KUKA KRL program: EPS_2_25252_SD6A_A_20250910061730.src

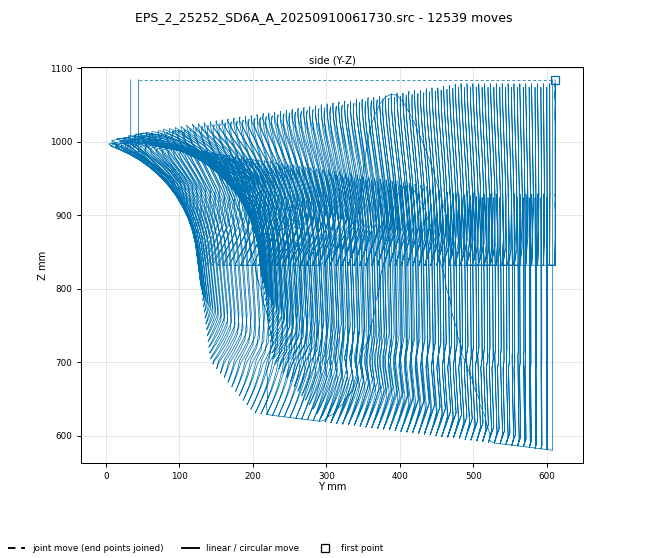
[picture p0: tool path of EPS_2_25252_SD6A_A_20250910061730.src, 12539 of 12541 moves have a stored position in this frame; points joined in program order, loops and branches not executed]
&ACCESS RVP
&REL 4
&COMMENT QRS 19112012
&PARAM EDITMASK = *
DEF PART()
EXT BAS (BAS_COMMAND :IN,REAL :IN )
INT I
BAS (#INITMOV,0 )

;KUKA QRS Post kuka4.cps  Date:22-06-2017 !

File_ID=2826

QRS_PRE_INIT()

;Init var - Until changes are made in qrs_pre_init
Outlet_Square_prg=0
Inlet_1_Square_prg=0
Inlet_2_Square_prg=0
Inlet_3_Square_prg=0
Inlet_4_Square_prg=0
Inlet_5_Square_prg=0

Outlet_1={X 0.000, Y 484.060, Z 891.000, B 0.000, E1 0.000 }
Inlet_1={X 0.000, Y 511.230, Z 798.500, B 0.000, E1 160.000 }
Outlet_1_type=366
Inlet_1_type=201
;QRS#1=Sidecore dimensions
;QRS#2=375-15" PVC SDR 35
;QRS#3=200-8" PVC SDR 35
;QRS#4=
;QRS#5=
;QRS#6=
;QRS#7=
;QRS#8=
;QRS#9=20Y PSX
;QRS#10=12-08 PSX
;QRS#11=
;QRS#12=
;QRS#13=
;QRS#14=
;QRS#15=
;QRS#16=1220x127x1372 4,5'
;QRS#17=EPS Height
;QRS#18=1074
;QRS#19=*
;QRS#20= UPDATED VERSION 22-06-2017
;QRS#21=*
Outlet_Square=0250
Inlet_1_Square=0100
Inlet_2_Square=0
Inlet_3_Square=0
Inlet_4_Square=0
Inlet_5_Square=0
Mill_Square=1
Outlet_Square_Prg=252
Inlet_1_Square_prg=204

QRS_INIT()

$ADVANCE=5

; T1
PTP {E1 177.357,E2 177.357}
PTP {X 0,Y 611.096,A -85,B 0,C 180,E1 177.357,E2 177.357,E3 0,E4 0,E5 0,E6 0}
QRS_SPEED_INIT()
LIN {X 0,Y 611.096,Z 1084,A -85,B 0,C 180,E1 177.357,E2 177.357,E3 0,E4 0,E5 0,E6 0} C_VEL
LIN {X 0,Y 611.096,Z 833.81,A -85,B 0,C 180,E1 177.357,E2 177.357} C_VEL
LIN {X 0,Y 611.169,Z 831.81,A -85,B 0,C 180,E1 177.544,E2 177.544} C_VEL
LIN {X 0,Y 611.846,Z 831.81,A -85,B 0,C 180,E1 178.833,E2 178.833} C_VEL
LIN {X 0,Y 611.842,Z 831.81,A -85,B 0,C 180,E1 185.845,E2 185.845} C_VEL
LIN {X 0,Y 611.87,Z 831.81,A -85,B 0,C 180,E1 192.946,E2 192.946} C_VEL
LIN {X 0,Y 611.805,Z 831.81,A -85,B 0,C 180,E1 200.259,E2 200.259} C_VEL
LIN {X 0,Y 611.785,Z 831.81,A -85,B 0,C 180,E1 207.936,E2 207.936} C_VEL
LIN {X 0,Y 610.448,Z 831.81,A -85,B 0,C 180,E1 210.686,E2 210.686} C_VEL
LIN {X 0,Y 611.751,Z 831.81,A -85,B 0,C 180,E1 216.209,E2 216.209} C_VEL
LIN {X 0,Y 611.181,Z 831.81,A -85,B 0,C 180,E1 217.329,E2 217.329} C_VEL
LIN {X 0,Y 610.711,Z 831.81,A -85,B 0,C 180,E1 222.327,E2 222.327} C_VEL
LIN {X 0,Y 611.733,Z 831.81,A -85,B 0,C 180,E1 224.523,E2 224.523} C_VEL
LIN {X 0,Y 611.705,Z 831.81,A -85,B 0,C 180,E1 232.607,E2 232.607} C_VEL
LIN {X 0,Y 611.184,Z 831.81,A -85,B 0,C 180,E1 233.752,E2 233.752} C_VEL
LIN {X 0,Y 611.693,Z 831.81,A -85,B 0,C 180,E1 241.163,E2 241.163} C_VEL
LIN {X 0,Y 611.503,Z 831.81,A -85,B 0,C 180,E1 242.05,E2 242.05} C_VEL
LIN {X 0,Y 611.8,Z 831.81,A -85,B 0,C 180,E1 248.625,E2 248.625} C_VEL
LIN {X 0,Y 610.992,Z 831.81,A -85,B 0,C 180,E1 248.983,E2 248.983} C_VEL
LIN {X 0,Y 610.765,Z 831.863,A -85,B 0,C 180,E1 249.009,E2 249.009} C_VEL
LIN {X 0,Y 611.59,Z 868.04,A -85,B 0,C 180,E1 249.483,E2 249.483} C_VEL
LIN {X 0,Y 611.819,Z 897.067,A -85,B 0,C 180,E1 249.858,E2 249.858} C_VEL
LIN {X 0,Y 611.837,Z 906.232,A -85,B 0,C 180,E1 250.014,E2 250.014} C_VEL
LIN {X 0,Y 611.813,Z 915.284,A -85,B 0,C 180,E1 250.207,E2 250.207} C_VEL
LIN {X 0,Y 611.665,Z 924.239,A -85,B 0,C 180,E1 250.435,E2 250.435} C_VEL
LIN {X 0,Y 611.793,Z 933.099,A -85,B 0,C 180,E1 250.71,E2 250.71} C_VEL
LIN {X 0,Y 611.793,Z 940.863,A -85,B 0,C 180,E1 250.98,E2 250.98} C_VEL
LIN {X 0,Y 611.788,Z 950.494,A -85,B 0,C 180,E1 251.365,E2 251.365} C_VEL
LIN {X 0,Y 611.804,Z 958.998,A -85,B 0,C 180,E1 251.75,E2 251.75} C_VEL
LIN {X 0,Y 611.728,Z 968.053,A -85,B 0,C 180,E1 252.208,E2 252.208} C_VEL
LIN {X 0,Y 611.708,Z 977.508,A -85,B 0,C 180,E1 252.747,E2 252.747} C_VEL
LIN {X 0,Y 611.545,Z 985.953,A -85,B 0,C 180,E1 253.278,E2 253.278} C_VEL
LIN {X 0,Y 611.448,Z 992.373,A -85,B 0,C 180,E1 253.719,E2 253.719} C_VEL
LIN {X 0,Y 611.514,Z 999.796,A -85,B 0,C 180,E1 254.279,E2 254.279} C_VEL
LIN {X 0,Y 611.73,Z 1007.694,A -85,B 0,C 180,E1 254.936,E2 254.936} C_VEL
LIN {X 0,Y 611.83,Z 1014.191,A -85,B 0,C 180,E1 255.523,E2 255.523} C_VEL
LIN {X 0,Y 611.643,Z 1021.1,A -85,B 0,C 180,E1 256.197,E2 256.197} C_VEL
LIN {X 0,Y 611.384,Z 1027.094,A -85,B 0,C 180,E1 256.831,E2 256.831} C_VEL
LIN {X 0,Y 611.257,Z 1032.807,A -85,B 0,C 180,E1 257.49,E2 257.49} C_VEL
LIN {X 0,Y 611.362,Z 1038.701,A -85,B 0,C 180,E1 258.239,E2 258.239} C_VEL
LIN {X 0,Y 611.558,Z 1043.069,A -85,B 0,C 180,E1 258.838,E2 258.838} C_VEL
LIN {X 0,Y 611.864,Z 1048.943,A -85,B 0,C 180,E1 259.735,E2 259.735} C_VEL
LIN {X 0,Y 611.485,Z 1054.185,A -85,B 0,C 180,E1 260.617,E2 260.617} C_VEL
LIN {X 0,Y 611.212,Z 1057.398,A -85,B 0,C 180,E1 261.204,E2 261.204} C_VEL
LIN {X 0,Y 611.06,Z 1061.684,A -85,B 0,C 180,E1 262.088,E2 262.088} C_VEL
LIN {X 0,Y 611.227,Z 1065.436,A -85,B 0,C 180,E1 262.974,E2 262.974} C_VEL
LIN {X 0,Y 611.629,Z 1068.68,A -85,B 0,C 180,E1 263.86,E2 263.86} C_VEL
LIN {X 0,Y 611.768,Z 1069.615,A -85,B 0,C 180,E1 264.154,E2 264.154} C_VEL
LIN {X 0,Y 611.736,Z 1071.453,A -85,B 0,C 180,E1 264.74,E2 264.74} C_VEL
LIN {X 0,Y 611.169,Z 1074.43,A -85,B 0,C 180,E1 265.908,E2 265.908} C_VEL
LIN {X 0,Y 610.975,Z 1075.682,A -85,B 0,C 180,E1 266.492,E2 266.492} C_VEL
LIN {X 0,Y 611.094,Z 1077.535,A -85,B 0,C 180,E1 267.712,E2 267.712} C_VEL
LIN {X 0,Y 611.599,Z 1078.552,A -85,B 0,C 180,E1 268.833,E2 268.833} C_VEL
LIN {X 0,Y 611.822,Z 1078.786,A -85,B 0,C 180,E1 269.3,E2 269.3} C_VEL
LIN {X 0,Y 611.469,Z 1078.916,A -85,B 0,C 180,E1 270.234,E2 270.234} C_VEL
LIN {X 0,Y 611.076,Z 1078.575,A -85,B 0,C 180,E1 271.168,E2 271.168} C_VEL
LIN {X 0,Y 611.004,Z 1077.586,A -85,B 0,C 180,E1 272.247,E2 272.247} C_VEL
LIN {X 0,Y 611.445,Z 1075.667,A -85,B 0,C 180,E1 273.505,E2 273.505} C_VEL
LIN {X 0,Y 611.741,Z 1074.409,A -85,B 0,C 180,E1 274.088,E2 274.088} C_VEL
LIN {X 0,Y 611.75,Z 1073.023,A -85,B 0,C 180,E1 274.674,E2 274.674} C_VEL
LIN {X 0,Y 611.456,Z 1071.462,A -85,B 0,C 180,E1 275.262,E2 275.262} C_VEL
LIN {X 0,Y 611.035,Z 1068.69,A -85,B 0,C 180,E1 276.146,E2 276.146} C_VEL
LIN {X 0,Y 610.903,Z 1065.436,A -85,B 0,C 180,E1 277.03,E2 277.03} C_VEL
LIN {X 0,Y 611.131,Z 1061.684,A -85,B 0,C 180,E1 277.911,E2 277.911} C_VEL
LIN {X 0,Y 611.584,Z 1057.398,A -85,B 0,C 180,E1 278.79,E2 278.79} C_VEL
LIN {X 0,Y 611.866,Z 1054.185,A -85,B 0,C 180,E1 279.377,E2 279.377} C_VEL
LIN {X 0,Y 611.514,Z 1048.943,A -85,B 0,C 180,E1 280.271,E2 280.271} C_VEL
LIN {X 0,Y 611.151,Z 1041.996,A -85,B 0,C 180,E1 281.318,E2 281.318} C_VEL
LIN {X 0,Y 611.162,Z 1036.427,A -85,B 0,C 180,E1 282.063,E2 282.063} C_VEL
LIN {X 0,Y 611.413,Z 1030.293,A -85,B 0,C 180,E1 282.806,E2 282.806} C_VEL
LIN {X 0,Y 611.786,Z 1022.804,A -85,B 0,C 180,E1 283.623,E2 283.623} C_VEL
LIN {X 0,Y 611.786,Z 1016.857,A -85,B 0,C 180,E1 284.223,E2 284.223} C_VEL
LIN {X 0,Y 611.564,Z 1009.74,A -85,B 0,C 180,E1 284.888,E2 284.888} C_VEL
LIN {X 0,Y 611.414,Z 1003.125,A -85,B 0,C 180,E1 285.456,E2 285.456} C_VEL
LIN {X 0,Y 611.434,Z 996.152,A -85,B 0,C 180,E1 286.003,E2 286.003} C_VEL
LIN {X 0,Y 611.593,Z 988.528,A -85,B 0,C 180,E1 286.547,E2 286.547} C_VEL
LIN {X 0,Y 611.77,Z 980.343,A -85,B 0,C 180,E1 287.078,E2 287.078} C_VEL
LIN {X 0,Y 611.808,Z 972.308,A -85,B 0,C 180,E1 287.555,E2 287.555} C_VEL
LIN {X 0,Y 611.781,Z 963.646,A -85,B 0,C 180,E1 288.02,E2 288.02} C_VEL
LIN {X 0,Y 611.699,Z 955.729,A -85,B 0,C 180,E1 288.407,E2 288.407} C_VEL
LIN {X 0,Y 611.702,Z 946.825,A -85,B 0,C 180,E1 288.792,E2 288.792} C_VEL
LIN {X 0,Y 611.79,Z 936.538,A -85,B 0,C 180,E1 289.174,E2 289.174} C_VEL
LIN {X 0,Y 611.757,Z 926.929,A -85,B 0,C 180,E1 289.485,E2 289.485} C_VEL
LIN {X 0,Y 611.762,Z 920.133,A -85,B 0,C 180,E1 289.678,E2 289.678} C_VEL
LIN {X 0,Y 611.841,Z 908.254,A -85,B 0,C 180,E1 289.947,E2 289.947} C_VEL
LIN {X 0,Y 611.832,Z 898.402,A -85,B 0,C 180,E1 290.122,E2 290.122} C_VEL
LIN {X 0,Y 611.682,Z 875.23,A -85,B 0,C 180,E1 290.425,E2 290.425} C_VEL
LIN {X 0,Y 610.968,Z 838.514,A -85,B 0,C 180,E1 290.902,E2 290.902} C_VEL
LIN {X 0,Y 610.816,Z 831.81,A -85,B 0,C 180,E1 290.998,E2 290.998} C_VEL
LIN {X 0,Y 611.657,Z 831.81,A -85,B 0,C 180,E1 291.131,E2 291.131} C_VEL
LIN {X 0,Y 611.596,Z 831.81,A -85,B 0,C 180,E1 291.733,E2 291.733} C_VEL
LIN {X 0,Y 611.82,Z 831.81,A -85,B 0,C 180,E1 297.934,E2 297.934} C_VEL
LIN {X 0,Y 610.469,Z 831.81,A -85,B 0,C 180,E1 300.685,E2 300.685} C_VEL
LIN {X 0,Y 611.751,Z 831.81,A -85,B 0,C 180,E1 306.209,E2 306.209} C_VEL
LIN {X 0,Y 611.184,Z 831.81,A -85,B 0,C 180,E1 307.329,E2 307.329} C_VEL
LIN {X 0,Y 610.712,Z 831.81,A -85,B 0,C 180,E1 312.326,E2 312.326} C_VEL
LIN {X 0,Y 611.746,Z 831.81,A -85,B 0,C 180,E1 314.524,E2 314.524} C_VEL
LIN {X 0,Y 611.724,Z 831.81,A -85,B 0,C 180,E1 322.605,E2 322.605} C_VEL
LIN {X 0,Y 611.197,Z 831.81,A -85,B 0,C 180,E1 323.753,E2 323.753} C_VEL
LIN {X 0,Y 611.636,Z 831.81,A -85,B 0,C 180,E1 331.172,E2 331.172} C_VEL
LIN {X 0,Y 611.414,Z 831.81,A -85,B 0,C 180,E1 332.046,E2 332.046} C_VEL
LIN {X 0,Y 611.821,Z 831.81,A -85,B 0,C 180,E1 339.742,E2 339.742} C_VEL
LIN {X 0,Y 611.864,Z 831.81,A -85,B 0,C 180,E1 347.054,E2 347.054} C_VEL
LIN {X 0,Y 611.851,Z 831.81,A -85,B 0,C 180,E1 354.155,E2 354.155} C_VEL
LIN {X 0,Y 611.852,Z 831.81,A -85,B 0,C 180,E1 361.167,E2 361.167} C_VEL
LIN {X 0,Y 611.868,Z 831.81,A -85,B 0,C 180,E1 368.196,E2 368.196} C_VEL
LIN {X 0,Y 611.822,Z 831.81,A -85,B 0,C 180,E1 375.354,E2 375.354} C_VEL
LIN {X 0,Y 611.846,Z 831.81,A -85,B 0,C 180,E1 382.766,E2 382.766} C_VEL
LIN {X 0,Y 611.833,Z 831.81,A -85,B 0,C 180,E1 390.609,E2 390.609} C_VEL
LIN {X 0,Y 611.787,Z 831.81,A -85,B 0,C 180,E1 399.156,E2 399.156} C_VEL
LIN {X 0,Y 610.375,Z 831.81,A -85,B 0,C 180,E1 402.355,E2 402.355} C_VEL
LIN {X 0,Y 610.682,Z 831.81,A -85,B 0,C 180,E1 405.577,E2 405.577} C_VEL
LIN {X 0,Y 611.77,Z 831.81,A -85,B 0,C 180,E1 407.764,E2 407.764} C_VEL
LIN {X 0,Y 610.278,Z 831.81,A -85,B 0,C 180,E1 413.69,E2 413.69} C_VEL
LIN {X 0,Y 611.794,Z 831.81,A -85,B 0,C 180,E1 416.636,E2 416.636} C_VEL
LIN {X 0,Y 611.82,Z 831.81,A -85,B 0,C 180,E1 424.677,E2 424.677} C_VEL
LIN {X 0,Y 611.504,Z 831.81,A -85,B 0,C 180,E1 433.291,E2 433.291} C_VEL
LIN {X 0,Y 611.274,Z 831.81,A -85,B 0,C 180,E1 434.632,E2 434.632} C_VEL
LIN {X 0,Y 611.861,Z 831.81,A -85,B 0,C 180,E1 441.804,E2 441.804} C_VEL
LIN {X 0,Y 611.873,Z 831.81,A -85,B 0,C 180,E1 448.833,E2 448.833} C_VEL
LIN {X 0,Y 611.827,Z 831.81,A -85,B 0,C 180,E1 457.977,E2 457.977} C_VEL
LIN {X 0,Y 611.67,Z 831.824,A -85,B 0,C 180,E1 458.051,E2 458.051} C_VEL
LIN {X 0,Y 611.815,Z 840.522,A -85,B 0,C 180,E1 458.307,E2 458.307} C_VEL
LIN {X 0,Y 611.718,Z 847.873,A -85,B 0,C 180,E1 458.567,E2 458.567} C_VEL
LIN {X 0,Y 611.699,Z 856.418,A -85,B 0,C 180,E1 458.936,E2 458.936} C_VEL
LIN {X 0,Y 611.782,Z 863.62,A -85,B 0,C 180,E1 459.304,E2 459.304} C_VEL
LIN {X 0,Y 611.819,Z 871.1,A -85,B 0,C 180,E1 459.748,E2 459.748} C_VEL
LIN {X 0,Y 611.737,Z 877.656,A -85,B 0,C 180,E1 460.193,E2 460.193} C_VEL
LIN {X 0,Y 611.613,Z 882.484,A -85,B 0,C 180,E1 460.566,E2 460.566} C_VEL
LIN {X 0,Y 611.52,Z 887.919,A -85,B 0,C 180,E1 461.014,E2 461.014} C_VEL
LIN {X 0,Y 611.753,Z 896.902,A -85,B 0,C 180,E1 461.902,E2 461.902} C_VEL
LIN {X 0,Y 611.846,Z 902.025,A -85,B 0,C 180,E1 462.498,E2 462.498} C_VEL
LIN {X 0,Y 611.57,Z 907.062,A -85,B 0,C 180,E1 463.155,E2 463.155} C_VEL
LIN {X 0,Y 611.352,Z 911.117,A -85,B 0,C 180,E1 463.768,E2 463.768} C_VEL
LIN {X 0,Y 611.348,Z 914.59,A -85,B 0,C 180,E1 464.365,E2 464.365} C_VEL
LIN {X 0,Y 611.521,Z 917.619,A -85,B 0,C 180,E1 464.961,E2 464.961} C_VEL
LIN {X 0,Y 611.856,Z 920.987,A -85,B 0,C 180,E1 465.746,E2 465.746} C_VEL
LIN {X 0,Y 611.761,Z 922.47,A -85,B 0,C 180,E1 466.142,E2 466.142} C_VEL
LIN {X 0,Y 611.48,Z 924.28,A -85,B 0,C 180,E1 466.702,E2 466.702} C_VEL
LIN {X 0,Y 611.285,Z 925.515,A -85,B 0,C 180,E1 467.157,E2 467.157} C_VEL
LIN {X 0,Y 611.186,Z 926.958,A -85,B 0,C 180,E1 467.808,E2 467.808} C_VEL
LIN {X 0,Y 611.315,Z 927.93,A -85,B 0,C 180,E1 468.419,E2 468.419} C_VEL
LIN {X 0,Y 611.592,Z 928.562,A -85,B 0,C 180,E1 469.026,E2 469.026} C_VEL
LIN {X 0,Y 611.86,Z 928.874,A -85,B 0,C 180,E1 469.636,E2 469.636} C_VEL
LIN {X 0,Y 611.627,Z 928.89,A -85,B 0,C 180,E1 470.265,E2 470.265} C_VEL
LIN {X 0,Y 611.328,Z 928.619,A -85,B 0,C 180,E1 470.822,E2 470.822} C_VEL
LIN {X 0,Y 611.148,Z 928.071,A -85,B 0,C 180,E1 471.378,E2 471.378} C_VEL
LIN {X 0,Y 611.15,Z 926.993,A -85,B 0,C 180,E1 472.083,E2 472.083} C_VEL
LIN {X 0,Y 611.421,Z 925.429,A -85,B 0,C 180,E1 472.783,E2 472.783} C_VEL
LIN {X 0,Y 611.841,Z 923.085,A -85,B 0,C 180,E1 473.578,E2 473.578} C_VEL
LIN {X 0,Y 611.756,Z 921.443,A -85,B 0,C 180,E1 474.044,E2 474.044} C_VEL
LIN {X 0,Y 611.36,Z 917.799,A -85,B 0,C 180,E1 474.914,E2 474.914} C_VEL
LIN {X 0,Y 611.233,Z 914.497,A -85,B 0,C 180,E1 475.563,E2 475.563} C_VEL
LIN {X 0,Y 611.356,Z 910.756,A -85,B 0,C 180,E1 476.201,E2 476.201} C_VEL
LIN {X 0,Y 611.663,Z 906.487,A -85,B 0,C 180,E1 476.834,E2 476.834} C_VEL
LIN {X 0,Y 611.852,Z 903.246,A -85,B 0,C 180,E1 477.263,E2 477.263} C_VEL
LIN {X 0,Y 611.704,Z 897.513,A -85,B 0,C 180,E1 477.94,E2 477.94} C_VEL
LIN {X 0,Y 611.516,Z 891.281,A -85,B 0,C 180,E1 478.574,E2 478.574} C_VEL
LIN {X 0,Y 611.48,Z 886.829,A -85,B 0,C 180,E1 478.988,E2 478.988} C_VEL
LIN {X 0,Y 611.701,Z 878.876,A -85,B 0,C 180,E1 479.63,E2 479.63} C_VEL
LIN {X 0,Y 611.854,Z 870.999,A -85,B 0,C 180,E1 480.168,E2 480.168} C_VEL
LIN {X 0,Y 611.776,Z 863.493,A -85,B 0,C 180,E1 480.613,E2 480.613} C_VEL
LIN {X 0,Y 611.65,Z 856.496,A -85,B 0,C 180,E1 480.971,E2 480.971} C_VEL
LIN {X 0,Y 611.658,Z 848.88,A -85,B 0,C 180,E1 481.306,E2 481.306} C_VEL
LIN {X 0,Y 611.817,Z 840.491,A -85,B 0,C 180,E1 481.604,E2 481.604} C_VEL
LIN {X 0,Y 611.738,Z 831.81,A -85,B 0,C 180,E1 481.86,E2 481.86} C_VEL
LIN {X 0,Y 611.761,Z 831.81,A -85,B 0,C 180,E1 489.158,E2 489.158} C_VEL
LIN {X 0,Y 610.343,Z 831.81,A -85,B 0,C 180,E1 492.358,E2 492.358} C_VEL
LIN {X 0,Y 610.656,Z 831.81,A -85,B 0,C 180,E1 495.58,E2 495.58} C_VEL
LIN {X 0,Y 611.745,Z 831.81,A -85,B 0,C 180,E1 497.762,E2 497.762} C_VEL
LIN {X 0,Y 611.804,Z 831.81,A -85,B 0,C 180,E1 506.626,E2 506.626} C_VEL
LIN {X 0,Y 611.798,Z 831.81,A -85,B 0,C 180,E1 514.676,E2 514.676} C_VEL
LIN {X 0,Y 611.517,Z 831.81,A -85,B 0,C 180,E1 523.287,E2 523.287} C_VEL
LIN {X 0,Y 611.274,Z 831.81,A -85,B 0,C 180,E1 524.632,E2 524.632} C_VEL
LIN {X 0,Y 611.874,Z 831.81,A -85,B 0,C 180,E1 531.804,E2 531.804} C_VEL
LIN {X 0,Y 611.169,Z 831.81,A -85,B 0,C 180,E1 537.544,E2 537.544} C_VEL
LIN {X 0,Y 602.919,Z 831.81,A -85,B 0,C 180,E1 540.819,E2 540.819} C_VEL
LIN {X 0,Y 602.895,Z 831.81,A -85,B 0,C 180,E1 547.96,E2 547.96} C_VEL
LIN {X 0,Y 602.752,Z 831.81,A -85,B 0,C 180,E1 555.331,E2 555.331} C_VEL
LIN {X 0,Y 603.111,Z 831.81,A -85,B 0,C 180,E1 561.401,E2 561.401} C_VEL
LIN {X 0,Y 602.758,Z 831.81,A -85,B 0,C 180,E1 569.705,E2 569.705} C_VEL
LIN {X 0,Y 603.046,Z 831.81,A -85,B 0,C 180,E1 577.563,E2 577.563} C_VEL
LIN {X 0,Y 602.75,Z 831.81,A -85,B 0,C 180,E1 586.183,E2 586.183} C_VEL
LIN {X 0,Y 603.17,Z 831.81,A -85,B 0,C 180,E1 593.755,E2 593.755} C_VEL
LIN {X 0,Y 603.374,Z 831.81,A -85,B 0,C 180,E1 602.271,E2 602.271} C_VEL
LIN {X 0,Y 603.327,Z 833.276,A -85,B 0,C 180,E1 608.755,E2 608.755} C_VEL
LIN {X 0,Y 604.135,Z 926.855,A -85,B 0,C 180,E1 610.257,E2 610.257} C_VEL
LIN {X 0,Y 603.999,Z 977.952,A -85,B 0,C 180,E1 612.547,E2 612.547} C_VEL
LIN {X 0,Y 603.794,Z 1020.941,A -85,B 0,C 180,E1 615.997,E2 615.997} C_VEL
LIN {X 0,Y 603.674,Z 1052.748,A -85,B 0,C 180,E1 620.231,E2 620.231} C_VEL
LIN {X 0,Y 603.605,Z 1072.224,A -85,B 0,C 180,E1 624.952,E2 624.952} C_VEL
LIN {X 0,Y 603.823,Z 1078.839,A -85,B 0,C 180,E1 629.28,E2 629.28} C_VEL
LIN {X 0,Y 603.745,Z 1074.049,A -85,B 0,C 180,E1 634.325,E2 634.325} C_VEL
LIN {X 0,Y 603.912,Z 1054.728,A -85,B 0,C 180,E1 639.401,E2 639.401} C_VEL
LIN {X 0,Y 603.891,Z 1022.734,A -85,B 0,C 180,E1 643.812,E2 643.812} C_VEL
LIN {X 0,Y 604.054,Z 979.467,A -85,B 0,C 180,E1 647.358,E2 647.358} C_VEL
LIN {X 0,Y 604.208,Z 927.768,A -85,B 0,C 180,E1 649.714,E2 649.714} C_VEL
LIN {X 0,Y 603.614,Z 844.819,A -85,B 0,C 180,E1 651.09,E2 651.09} C_VEL
LIN {X 0,Y 603.646,Z 831.81,A -85,B 0,C 180,E1 651.379,E2 651.379} C_VEL
LIN {X 0,Y 602.798,Z 831.81,A -85,B 0,C 180,E1 659.702,E2 659.702} C_VEL
LIN {X 0,Y 603.057,Z 831.81,A -85,B 0,C 180,E1 667.558,E2 667.558} C_VEL
LIN {X 0,Y 602.765,Z 831.81,A -85,B 0,C 180,E1 676.178,E2 676.178} C_VEL
LIN {X 0,Y 603.197,Z 831.81,A -85,B 0,C 180,E1 683.752,E2 683.752} C_VEL
LIN {X 0,Y 603.265,Z 831.81,A -85,B 0,C 180,E1 692.262,E2 692.262} C_VEL
LIN {X 0,Y 602.872,Z 831.81,A -85,B 0,C 180,E1 701.658,E2 701.658} C_VEL
LIN {X 0,Y 602.912,Z 831.81,A -85,B 0,C 180,E1 709.116,E2 709.116} C_VEL
LIN {X 0,Y 602.859,Z 831.81,A -85,B 0,C 180,E1 716.39,E2 716.39} C_VEL
LIN {X 0,Y 602.818,Z 831.81,A -85,B 0,C 180,E1 723.607,E2 723.607} C_VEL
LIN {X 0,Y 603.208,Z 831.81,A -85,B 0,C 180,E1 729.411,E2 729.411} C_VEL
LIN {X 0,Y 603.025,Z 831.81,A -85,B 0,C 180,E1 736.822,E2 736.822} C_VEL
LIN {X 0,Y 602.843,Z 831.81,A -85,B 0,C 180,E1 744.542,E2 744.542} C_VEL
LIN {X 0,Y 602.661,Z 831.81,A -85,B 0,C 180,E1 752.482,E2 752.482} C_VEL
LIN {X 0,Y 603.278,Z 831.81,A -85,B 0,C 180,E1 759.901,E2 759.901} C_VEL
LIN {X 0,Y 603.426,Z 831.81,A -85,B 0,C 180,E1 768.207,E2 768.207} C_VEL
LIN {X 0,Y 603.275,Z 831.81,A -85,B 0,C 180,E1 777.428,E2 777.428} C_VEL
LIN {X 0,Y 603.196,Z 831.81,A -85,B 0,C 180,E1 785.473,E2 785.473} C_VEL
LIN {X 0,Y 603.241,Z 831.81,A -85,B 0,C 180,E1 794.684,E2 794.684} C_VEL
LIN {X 0,Y 602.911,Z 831.81,A -85,B 0,C 180,E1 803.857,E2 803.857} C_VEL
LIN {X 0,Y 602.597,Z 831.81,A -85,B 0,C 180,E1 810.721,E2 810.721} C_VEL
LIN {X 0,Y 603.88,Z 833.613,A -85,B 0,C 180,E1 817.944,E2 817.944} C_VEL
LIN {X 0,Y 603.909,Z 873.408,A -85,B 0,C 180,E1 819.765,E2 819.765} C_VEL
LIN {X 0,Y 603.782,Z 904.415,A -85,B 0,C 180,E1 822.704,E2 822.704} C_VEL
LIN {X 0,Y 603.602,Z 923.583,A -85,B 0,C 180,E1 826.43,E2 826.43} C_VEL
LIN {X 0,Y 603.782,Z 928.979,A -85,B 0,C 180,E1 829.834,E2 829.834} C_VEL
LIN {X 0,Y 603.782,Z 922.083,A -85,B 0,C 180,E1 833.931,E2 833.931} C_VEL
LIN {X 0,Y 603.79,Z 900.446,A -85,B 0,C 180,E1 837.708,E2 837.708} C_VEL
LIN {X 0,Y 603.924,Z 866.99,A -85,B 0,C 180,E1 840.551,E2 840.551} C_VEL
LIN {X 0,Y 603.555,Z 831.81,A -85,B 0,C 180,E1 842.136,E2 842.136} C_VEL
LIN {X 0,Y 603.276,Z 831.81,A -85,B 0,C 180,E1 849.9,E2 849.9} C_VEL
LIN {X 0,Y 603.388,Z 831.81,A -85,B 0,C 180,E1 858.203,E2 858.203} C_VEL
LIN {X 0,Y 603.273,Z 831.81,A -85,B 0,C 180,E1 867.425,E2 867.425} C_VEL
LIN {X 0,Y 603.205,Z 831.81,A -85,B 0,C 180,E1 875.474,E2 875.474} C_VEL
LIN {X 0,Y 603.234,Z 831.81,A -85,B 0,C 180,E1 884.684,E2 884.684} C_VEL
LIN {X 0,Y 602.924,Z 831.81,A -85,B 0,C 180,E1 893.824,E2 893.824} C_VEL
LIN {X 0,Y 602.919,Z 831.81,A -85,B 0,C 180,E1 900.819,E2 900.819} C_VEL
LIN {X 0,Y 594.992,Z 831.81,A -85,B 0,C 180,E1 904.119,E2 904.119} C_VEL
LIN {X 0,Y 595.477,Z 831.81,A -85,B 0,C 180,E1 912.513,E2 912.513} C_VEL
LIN {X 0,Y 594.993,Z 831.81,A -85,B 0,C 180,E1 921.708,E2 921.708} C_VEL
LIN {X 0,Y 594.722,Z 831.81,A -85,B 0,C 180,E1 929.843,E2 929.843} C_VEL
LIN {X 0,Y 595.417,Z 831.81,A -85,B 0,C 180,E1 936.799,E2 936.799} C_VEL
LIN {X 0,Y 595.012,Z 831.81,A -85,B 0,C 180,E1 945.463,E2 945.463} C_VEL
LIN {X 0,Y 595.231,Z 831.81,A -85,B 0,C 180,E1 953.433,E2 953.433} C_VEL
LIN {X 0,Y 595.314,Z 831.81,A -85,B 0,C 180,E1 961.863,E2 961.863} C_VEL
LIN {X 0,Y 595.572,Z 832.317,A -85,B 0,C 180,E1 968.453,E2 968.453} C_VEL
LIN {X 0,Y 596.6,Z 925.857,A -85,B 0,C 180,E1 969.968,E2 969.968} C_VEL
LIN {X 0,Y 596.264,Z 978.236,A -85,B 0,C 180,E1 972.331,E2 972.331} C_VEL
LIN {X 0,Y 595.889,Z 1022.739,A -85,B 0,C 180,E1 976,E2 976} C_VEL
LIN {X 0,Y 595.564,Z 1054.732,A -85,B 0,C 180,E1 980.467,E2 980.467} C_VEL
LIN {X 0,Y 595.294,Z 1074.051,A -85,B 0,C 180,E1 985.614,E2 985.614} C_VEL
LIN {X 0,Y 595.235,Z 1078.839,A -85,B 0,C 180,E1 990.731,E2 990.731} C_VEL
LIN {X 0,Y 595.294,Z 1070.858,A -85,B 0,C 180,E1 995.615,E2 995.615} C_VEL
LIN {X 0,Y 595.497,Z 1048.376,A -85,B 0,C 180,E1 1000.647,E2 1000.647} C_VEL
LIN {X 0,Y 595.913,Z 1013.07,A -85,B 0,C 180,E1 1004.983,E2 1004.983} C_VEL
LIN {X 0,Y 596.426,Z 966.403,A -85,B 0,C 180,E1 1008.357,E2 1008.357} C_VEL
LIN {X 0,Y 596.776,Z 914.035,A -85,B 0,C 180,E1 1010.344,E2 1010.344} C_VEL
LIN {X 0,Y 595.497,Z 831.81,A -85,B 0,C 180,E1 1011.686,E2 1011.686} C_VEL
LIN {X 0,Y 594.76,Z 831.81,A -85,B 0,C 180,E1 1019.838,E2 1019.838} C_VEL
LIN {X 0,Y 595.413,Z 831.81,A -85,B 0,C 180,E1 1026.795,E2 1026.795} C_VEL
LIN {X 0,Y 595.023,Z 831.81,A -85,B 0,C 180,E1 1035.459,E2 1035.459} C_VEL
LIN {X 0,Y 595.252,Z 831.81,A -85,B 0,C 180,E1 1043.424,E2 1043.424} C_VEL
LIN {X 0,Y 595.212,Z 831.81,A -85,B 0,C 180,E1 1051.854,E2 1051.854} C_VEL
LIN {X 0,Y 594.959,Z 831.81,A -85,B 0,C 180,E1 1061.405,E2 1061.405} C_VEL
LIN {X 0,Y 594.922,Z 831.81,A -85,B 0,C 180,E1 1069.133,E2 1069.133} C_VEL
LIN {X 0,Y 594.87,Z 831.81,A -85,B 0,C 180,E1 1076.342,E2 1076.342} C_VEL
LIN {X 0,Y 594.808,Z 831.81,A -85,B 0,C 180,E1 1083.656,E2 1083.656} C_VEL
LIN {X 0,Y 594.773,Z 831.81,A -85,B 0,C 180,E1 1090.791,E2 1090.791} C_VEL
LIN {X 0,Y 594.954,Z 831.81,A -85,B 0,C 180,E1 1097.057,E2 1097.057} C_VEL
LIN {X 0,Y 594.671,Z 831.81,A -85,B 0,C 180,E1 1105.052,E2 1105.052} C_VEL
LIN {X 0,Y 595.187,Z 831.81,A -85,B 0,C 180,E1 1111.513,E2 1111.513} C_VEL
LIN {X 0,Y 594.686,Z 831.81,A -85,B 0,C 180,E1 1121.167,E2 1121.167} C_VEL
LIN {X 0,Y 594.696,Z 831.81,A -85,B 0,C 180,E1 1129.405,E2 1129.405} C_VEL
LIN {X 0,Y 594.776,Z 831.81,A -85,B 0,C 180,E1 1138.463,E2 1138.463} C_VEL
LIN {X 0,Y 594.505,Z 831.81,A -85,B 0,C 180,E1 1146.693,E2 1146.693} C_VEL
LIN {X 0,Y 595.241,Z 831.81,A -85,B 0,C 180,E1 1154.473,E2 1154.473} C_VEL
LIN {X 0,Y 595.046,Z 831.81,A -85,B 0,C 180,E1 1163.41,E2 1163.41} C_VEL
LIN {X 0,Y 594.587,Z 831.81,A -85,B 0,C 180,E1 1170.731,E2 1170.731} C_VEL
LIN {X 0,Y 595.811,Z 833.515,A -85,B 0,C 180,E1 1177.776,E2 1177.776} C_VEL
LIN {X 0,Y 596.011,Z 873.256,A -85,B 0,C 180,E1 1179.618,E2 1179.618} C_VEL
LIN {X 0,Y 595.814,Z 905.02,A -85,B 0,C 180,E1 1182.69,E2 1182.69} C_VEL
LIN {X 0,Y 595.501,Z 924.425,A -85,B 0,C 180,E1 1186.66,E2 1186.66} C_VEL
LIN {X 0,Y 595.63,Z 928.97,A -85,B 0,C 180,E1 1190.118,E2 1190.118} C_VEL
LIN {X 0,Y 595.655,Z 920.868,A -85,B 0,C 180,E1 1194.319,E2 1194.319} C_VEL
LIN {X 0,Y 595.755,Z 897.867,A -85,B 0,C 180,E1 1198.115,E2 1198.115} C_VEL
LIN {X 0,Y 595.988,Z 863.804,A -85,B 0,C 180,E1 1200.881,E2 1200.881} C_VEL
LIN {X 0,Y 595.43,Z 831.81,A -85,B 0,C 180,E1 1202.345,E2 1202.345} C_VEL
LIN {X 0,Y 594.667,Z 831.81,A -85,B 0,C 180,E1 1211.164,E2 1211.164} C_VEL
LIN {X 0,Y 594.647,Z 831.81,A -85,B 0,C 180,E1 1219.4,E2 1219.4} C_VEL
LIN {X 0,Y 594.776,Z 831.81,A -85,B 0,C 180,E1 1228.463,E2 1228.463} C_VEL
LIN {X 0,Y 594.494,Z 831.81,A -85,B 0,C 180,E1 1236.693,E2 1236.693} C_VEL
LIN {X 0,Y 595.238,Z 831.81,A -85,B 0,C 180,E1 1244.473,E2 1244.473} C_VEL
LIN {X 0,Y 595.062,Z 831.81,A -85,B 0,C 180,E1 1253.411,E2 1253.411} C_VEL
LIN {X 0,Y 594.937,Z 831.81,A -85,B 0,C 180,E1 1260.8,E2 1260.8} C_VEL
LIN {X 0,Y 594.992,Z 831.81,A -85,B 0,C 180,E1 1264.119,E2 1264.119} C_VEL
LIN {X 0,Y 587.053,Z 831.81,A -85,B 0,C 180,E1 1267.492,E2 1267.492} C_VEL
LIN {X 0,Y 587.151,Z 831.81,A -85,B 0,C 180,E1 1274.254,E2 1274.254} C_VEL
LIN {X 0,Y 586.857,Z 831.81,A -85,B 0,C 180,E1 1282.024,E2 1282.024} C_VEL
LIN {X 0,Y 586.571,Z 831.81,A -85,B 0,C 180,E1 1290.301,E2 1290.301} C_VEL
LIN {X 0,Y 586.838,Z 831.81,A -85,B 0,C 180,E1 1297.935,E2 1297.935} C_VEL
LIN {X 0,Y 586.545,Z 831.81,A -85,B 0,C 180,E1 1306.716,E2 1306.716} C_VEL
LIN {X 0,Y 586.734,Z 831.81,A -85,B 0,C 180,E1 1314.567,E2 1314.567} C_VEL
LIN {X 0,Y 586.93,Z 831.81,A -85,B 0,C 180,E1 1323.138,E2 1323.138} C_VEL
LIN {X 0,Y 587.57,Z 833.408,A -85,B 0,C 180,E1 1328.158,E2 1328.158} C_VEL
LIN {X 0,Y 589.069,Z 926.955,A -85,B 0,C 180,E1 1329.733,E2 1329.733} C_VEL
LIN {X 0,Y 588.573,Z 978.282,A -85,B 0,C 180,E1 1332.095,E2 1332.095} C_VEL
LIN {X 0,Y 588.04,Z 1022.739,A -85,B 0,C 180,E1 1335.809,E2 1335.809} C_VEL
LIN {X 0,Y 587.654,Z 1054.733,A -85,B 0,C 180,E1 1340.337,E2 1340.337} C_VEL
LIN {X 0,Y 587.323,Z 1074.051,A -85,B 0,C 180,E1 1345.555,E2 1345.555} C_VEL
LIN {X 0,Y 587.23,Z 1078.839,A -85,B 0,C 180,E1 1350.741,E2 1350.741} C_VEL
LIN {X 0,Y 587.257,Z 1070.683,A -85,B 0,C 180,E1 1355.749,E2 1355.749} C_VEL
LIN {X 0,Y 587.519,Z 1048.53,A -85,B 0,C 180,E1 1360.767,E2 1360.767} C_VEL
LIN {X 0,Y 588.044,Z 1012.95,A -85,B 0,C 180,E1 1365.2,E2 1365.2} C_VEL
LIN {X 0,Y 588.759,Z 966.478,A -85,B 0,C 180,E1 1368.601,E2 1368.601} C_VEL
LIN {X 0,Y 589.272,Z 914.553,A -85,B 0,C 180,E1 1370.602,E2 1370.602} C_VEL
LIN {X 0,Y 587.362,Z 831.81,A -85,B 0,C 180,E1 1372.002,E2 1372.002} C_VEL
LIN {X 0,Y 586.602,Z 831.81,A -85,B 0,C 180,E1 1380.296,E2 1380.296} C_VEL
LIN {X 0,Y 586.843,Z 831.81,A -85,B 0,C 180,E1 1387.928,E2 1387.928} C_VEL
LIN {X 0,Y 586.56,Z 831.81,A -85,B 0,C 180,E1 1396.712,E2 1396.712} C_VEL
LIN {X 0,Y 586.735,Z 831.81,A -85,B 0,C 180,E1 1404.56,E2 1404.56} C_VEL
LIN {X 0,Y 586.729,Z 831.81,A -85,B 0,C 180,E1 1413.167,E2 1413.167} C_VEL
LIN {X 0,Y 587.008,Z 831.81,A -85,B 0,C 180,E1 1421.144,E2 1421.144} C_VEL
LIN {X 0,Y 586.999,Z 831.81,A -85,B 0,C 180,E1 1428.818,E2 1428.818} C_VEL
LIN {X 0,Y 586.881,Z 831.81,A -85,B 0,C 180,E1 1436.292,E2 1436.292} C_VEL
LIN {X 0,Y 586.799,Z 831.81,A -85,B 0,C 180,E1 1443.706,E2 1443.706} C_VEL
LIN {X 0,Y 587.117,Z 831.81,A -85,B 0,C 180,E1 1449.671,E2 1449.671} C_VEL
LIN {X 0,Y 586.868,Z 831.81,A -85,B 0,C 180,E1 1457.299,E2 1457.299} C_VEL
LIN {X 0,Y 586.618,Z 831.81,A -85,B 0,C 180,E1 1465.267,E2 1465.267} C_VEL
LIN {X 0,Y 586.545,Z 831.81,A -85,B 0,C 180,E1 1472.769,E2 1472.769} C_VEL
LIN {X 0,Y 586.649,Z 831.81,A -85,B 0,C 180,E1 1481.273,E2 1481.273} C_VEL
LIN {X 0,Y 587.071,Z 831.81,A -85,B 0,C 180,E1 1488.764,E2 1488.764} C_VEL
LIN {X 0,Y 586.845,Z 831.81,A -85,B 0,C 180,E1 1497.986,E2 1497.986} C_VEL
LIN {X 0,Y 586.487,Z 831.81,A -85,B 0,C 180,E1 1506.721,E2 1506.721} C_VEL
LIN {X 0,Y 587.214,Z 831.81,A -85,B 0,C 180,E1 1514.255,E2 1514.255} C_VEL
LIN {X 0,Y 587.075,Z 831.81,A -85,B 0,C 180,E1 1523.32,E2 1523.32} C_VEL
LIN {X 0,Y 586.574,Z 831.81,A -85,B 0,C 180,E1 1530.741,E2 1530.741} C_VEL
LIN {X 0,Y 587.514,Z 832.544,A -85,B 0,C 180,E1 1537.574,E2 1537.574} C_VEL
LIN {X 0,Y 588.139,Z 873.092,A -85,B 0,C 180,E1 1539.467,E2 1539.467} C_VEL
LIN {X 0,Y 587.93,Z 904.247,A -85,B 0,C 180,E1 1542.484,E2 1542.484} C_VEL
LIN {X 0,Y 587.586,Z 924.031,A -85,B 0,C 180,E1 1546.479,E2 1546.479} C_VEL
LIN {X 0,Y 587.514,Z 928.904,A -85,B 0,C 180,E1 1550.408,E2 1550.408} C_VEL
LIN {X 0,Y 587.62,Z 920.768,A -85,B 0,C 180,E1 1554.406,E2 1554.406} C_VEL
LIN {X 0,Y 587.798,Z 898.641,A -85,B 0,C 180,E1 1558.136,E2 1558.136} C_VEL
LIN {X 0,Y 588.104,Z 863.998,A -85,B 0,C 180,E1 1561.019,E2 1561.019} C_VEL
LIN {X 0,Y 587.387,Z 831.81,A -85,B 0,C 180,E1 1562.412,E2 1562.412} C_VEL
LIN {X 0,Y 586.628,Z 831.81,A -85,B 0,C 180,E1 1571.273,E2 1571.273} C_VEL
LIN {X 0,Y 587.029,Z 831.81,A -85,B 0,C 180,E1 1578.76,E2 1578.76} C_VEL
LIN {X 0,Y 586.84,Z 831.81,A -85,B 0,C 180,E1 1587.986,E2 1587.986} C_VEL
LIN {X 0,Y 586.477,Z 831.81,A -85,B 0,C 180,E1 1596.719,E2 1596.719} C_VEL
LIN {X 0,Y 587.215,Z 831.81,A -85,B 0,C 180,E1 1604.256,E2 1604.256} C_VEL
LIN {X 0,Y 587.085,Z 831.81,A -85,B 0,C 180,E1 1613.321,E2 1613.321} C_VEL
LIN {X 0,Y 586.951,Z 831.81,A -85,B 0,C 180,E1 1620.742,E2 1620.742} C_VEL
LIN {X 0,Y 587.053,Z 831.81,A -85,B 0,C 180,E1 1627.492,E2 1627.492} C_VEL
LIN {X 0,Y 578.901,Z 831.81,A -85,B 0,C 180,E1 1630.883,E2 1630.883} C_VEL
LIN {X 0,Y 579.086,Z 831.81,A -85,B 0,C 180,E1 1639.124,E2 1639.124} C_VEL
LIN {X 0,Y 579.021,Z 831.81,A -85,B 0,C 180,E1 1649.007,E2 1649.007} C_VEL
LIN {X 0,Y 578.817,Z 831.81,A -85,B 0,C 180,E1 1658.038,E2 1658.038} C_VEL
LIN {X 0,Y 578.729,Z 831.81,A -85,B 0,C 180,E1 1666.151,E2 1666.151} C_VEL
LIN {X 0,Y 578.819,Z 831.81,A -85,B 0,C 180,E1 1673.85,E2 1673.85} C_VEL
LIN {X 0,Y 578.979,Z 831.81,A -85,B 0,C 180,E1 1682.698,E2 1682.698} C_VEL
LIN {X 0,Y 579.358,Z 833.175,A -85,B 0,C 180,E1 1687.829,E2 1687.829} C_VEL
LIN {X 0,Y 581.531,Z 926.094,A -85,B 0,C 180,E1 1689.432,E2 1689.432} C_VEL
LIN {X 0,Y 580.904,Z 977.959,A -85,B 0,C 180,E1 1691.829,E2 1691.829} C_VEL
LIN {X 0,Y 580.267,Z 1021.715,A -85,B 0,C 180,E1 1695.502,E2 1695.502} C_VEL
LIN {X 0,Y 579.715,Z 1054.733,A -85,B 0,C 180,E1 1700.204,E2 1700.204} C_VEL
LIN {X 0,Y 579.371,Z 1074.05,A -85,B 0,C 180,E1 1705.493,E2 1705.493} C_VEL
LIN {X 0,Y 579.239,Z 1078.839,A -85,B 0,C 180,E1 1710.751,E2 1710.751} C_VEL
LIN {X 0,Y 579.222,Z 1070.683,A -85,B 0,C 180,E1 1715.829,E2 1715.829} C_VEL
LIN {X 0,Y 579.51,Z 1047.863,A -85,B 0,C 180,E1 1721.03,E2 1721.03} C_VEL
LIN {X 0,Y 580.164,Z 1011.84,A -85,B 0,C 180,E1 1725.519,E2 1725.519} C_VEL
LIN {X 0,Y 581.128,Z 964.673,A -85,B 0,C 180,E1 1728.953,E2 1728.953} C_VEL
LIN {X 0,Y 581.835,Z 911.262,A -85,B 0,C 180,E1 1730.96,E2 1730.96} C_VEL
LIN {X 0,Y 579.299,Z 831.81,A -85,B 0,C 180,E1 1732.228,E2 1732.228} C_VEL
LIN {X 0,Y 578.462,Z 831.81,A -85,B 0,C 180,E1 1740.768,E2 1740.768} C_VEL
LIN {X 0,Y 578.821,Z 831.81,A -85,B 0,C 180,E1 1748.033,E2 1748.033} C_VEL
LIN {X 0,Y 578.74,Z 831.81,A -85,B 0,C 180,E1 1756.145,E2 1756.145} C_VEL
LIN {X 0,Y 578.824,Z 831.81,A -85,B 0,C 180,E1 1763.846,E2 1763.846} C_VEL
LIN {X 0,Y 578.802,Z 831.81,A -85,B 0,C 180,E1 1772.685,E2 1772.685} C_VEL
LIN {X 0,Y 579.096,Z 831.81,A -85,B 0,C 180,E1 1780.876,E2 1780.876} C_VEL
LIN {X 0,Y 578.82,Z 831.81,A -85,B 0,C 180,E1 1789.474,E2 1789.474} C_VEL
LIN {X 0,Y 578.916,Z 831.81,A -85,B 0,C 180,E1 1796.241,E2 1796.241} C_VEL
LIN {X 0,Y 578.82,Z 831.81,A -85,B 0,C 180,E1 1803.757,E2 1803.757} C_VEL
LIN {X 0,Y 578.867,Z 831.81,A -85,B 0,C 180,E1 1810.551,E2 1810.551} C_VEL
LIN {X 0,Y 578.812,Z 831.81,A -85,B 0,C 180,E1 1817.548,E2 1817.548} C_VEL
LIN {X 0,Y 578.542,Z 831.81,A -85,B 0,C 180,E1 1825.646,E2 1825.646} C_VEL
LIN {X 0,Y 578.643,Z 831.81,A -85,B 0,C 180,E1 1832.523,E2 1832.523} C_VEL
LIN {X 0,Y 578.548,Z 831.81,A -85,B 0,C 180,E1 1841.62,E2 1841.62} C_VEL
LIN {X 0,Y 578.442,Z 831.81,A -85,B 0,C 180,E1 1850.002,E2 1850.002} C_VEL
LIN {X 0,Y 578.67,Z 831.81,A -85,B 0,C 180,E1 1858.466,E2 1858.466} C_VEL
LIN {X 0,Y 578.706,Z 831.81,A -85,B 0,C 180,E1 1866.017,E2 1866.017} C_VEL
LIN {X 0,Y 578.765,Z 831.81,A -85,B 0,C 180,E1 1875.576,E2 1875.576} C_VEL
LIN {X 0,Y 579.095,Z 831.81,A -85,B 0,C 180,E1 1883.227,E2 1883.227} C_VEL
LIN {X 0,Y 578.561,Z 831.81,A -85,B 0,C 180,E1 1890.751,E2 1890.751} C_VEL
LIN {X 0,Y 579.542,Z 833.491,A -85,B 0,C 180,E1 1897.428,E2 1897.428} C_VEL
LIN {X 0,Y 580.223,Z 874.325,A -85,B 0,C 180,E1 1899.408,E2 1899.408} C_VEL
LIN {X 0,Y 579.833,Z 906.238,A -85,B 0,C 180,E1 1902.661,E2 1902.661} C_VEL
LIN {X 0,Y 579.579,Z 924.253,A -85,B 0,C 180,E1 1906.505,E2 1906.505} C_VEL
LIN {X 0,Y 579.426,Z 928.758,A -85,B 0,C 180,E1 1910.706,E2 1910.706} C_VEL
LIN {X 0,Y 579.405,Z 918.64,A -85,B 0,C 180,E1 1914.998,E2 1914.998} C_VEL
LIN {X 0,Y 579.778,Z 894.392,A -85,B 0,C 180,E1 1918.733,E2 1918.733} C_VEL
LIN {X 0,Y 580.208,Z 859.162,A -85,B 0,C 180,E1 1921.441,E2 1921.441} C_VEL
LIN {X 0,Y 579.258,Z 831.81,A -85,B 0,C 180,E1 1922.69,E2 1922.69} C_VEL
LIN {X 0,Y 578.528,Z 831.81,A -85,B 0,C 180,E1 1931.617,E2 1931.617} C_VEL
LIN {X 0,Y 578.384,Z 831.81,A -85,B 0,C 180,E1 1939.997,E2 1939.997} C_VEL
LIN {X 0,Y 578.666,Z 831.81,A -85,B 0,C 180,E1 1948.463,E2 1948.463} C_VEL
LIN {X 0,Y 578.699,Z 831.81,A -85,B 0,C 180,E1 1956.017,E2 1956.017} C_VEL
LIN {X 0,Y 578.754,Z 831.81,A -85,B 0,C 180,E1 1965.577,E2 1965.577} C_VEL
LIN {X 0,Y 579.104,Z 831.81,A -85,B 0,C 180,E1 1973.229,E2 1973.229} C_VEL
LIN {X 0,Y 578.971,Z 831.81,A -85,B 0,C 180,E1 1980.752,E2 1980.752} C_VEL
LIN {X 0,Y 578.831,Z 831.81,A -85,B 0,C 180,E1 1988.293,E2 1988.293} C_VEL
LIN {X 0,Y 578.901,Z 831.81,A -85,B 0,C 180,E1 1990.883,E2 1990.883} C_VEL
LIN {X 0,Y 571.066,Z 831.81,A -85,B 0,C 180,E1 1994.354,E2 1994.354} C_VEL
LIN {X 0,Y 570.664,Z 831.81,A -85,B 0,C 180,E1 2002.684,E2 2002.684} C_VEL
LIN {X 0,Y 570.593,Z 831.81,A -85,B 0,C 180,E1 2010.19,E2 2010.19} C_VEL
LIN {X 0,Y 570.61,Z 831.81,A -85,B 0,C 180,E1 2018.686,E2 2018.686} C_VEL
LIN {X 0,Y 570.381,Z 831.81,A -85,B 0,C 180,E1 2027.278,E2 2027.278} C_VEL
LIN {X 0,Y 570.444,Z 831.81,A -85,B 0,C 180,E1 2035.113,E2 2035.113} C_VEL
LIN {X 0,Y 570.73,Z 831.81,A -85,B 0,C 180,E1 2043.978,E2 2043.978} C_VEL
LIN {X 0,Y 571.296,Z 833.385,A -85,B 0,C 180,E1 2047.502,E2 2047.502} C_VEL
LIN {X 0,Y 574.329,Z 871.582,A -85,B 0,C 180,E1 2048.133,E2 2048.133} C_VEL
LIN {X 0,Y 574.01,Z 933.507,A -85,B 0,C 180,E1 2049.399,E2 2049.399} C_VEL
LIN {X 0,Y 573.051,Z 983.907,A -85,B 0,C 180,E1 2051.971,E2 2051.971} C_VEL
LIN {X 0,Y 572.213,Z 1026.182,A -85,B 0,C 180,E1 2055.8,E2 2055.8} C_VEL
LIN {X 0,Y 571.625,Z 1056.692,A -85,B 0,C 180,E1 2060.449,E2 2060.449} C_VEL
LIN {X 0,Y 571.392,Z 1074.05,A -85,B 0,C 180,E1 2065.43,E2 2065.43} C_VEL
LIN {X 0,Y 571.235,Z 1078.838,A -85,B 0,C 180,E1 2070.761,E2 2070.761} C_VEL
LIN {X 0,Y 571.155,Z 1070.117,A -85,B 0,C 180,E1 2076.101,E2 2076.101} C_VEL
LIN {X 0,Y 571.517,Z 1047.387,A -85,B 0,C 180,E1 2081.263,E2 2081.263} C_VEL
LIN {X 0,Y 572.327,Z 1011.488,A -85,B 0,C 180,E1 2085.771,E2 2085.771} C_VEL
LIN {X 0,Y 573.486,Z 964.676,A -85,B 0,C 180,E1 2089.215,E2 2089.215} C_VEL
LIN {X 0,Y 574.379,Z 911.261,A -85,B 0,C 180,E1 2091.245,E2 2091.245} C_VEL
LIN {X 0,Y 571.804,Z 834.8,A -85,B 0,C 180,E1 2092.458,E2 2092.458} C_VEL
LIN {X 0,Y 571.156,Z 831.81,A -85,B 0,C 180,E1 2092.66,E2 2092.66} C_VEL
LIN {X 0,Y 570.624,Z 831.81,A -85,B 0,C 180,E1 2100.186,E2 2100.186} C_VEL
LIN {X 0,Y 570.617,Z 831.81,A -85,B 0,C 180,E1 2108.681,E2 2108.681} C_VEL
LIN {X 0,Y 570.391,Z 831.81,A -85,B 0,C 180,E1 2117.273,E2 2117.273} C_VEL
LIN {X 0,Y 570.44,Z 831.81,A -85,B 0,C 180,E1 2125.108,E2 2125.108} C_VEL
LIN {X 0,Y 570.728,Z 831.81,A -85,B 0,C 180,E1 2132.968,E2 2132.968} C_VEL
LIN {X 0,Y 571.113,Z 831.81,A -85,B 0,C 180,E1 2140.613,E2 2140.613} C_VEL
LIN {X 0,Y 571.046,Z 831.81,A -85,B 0,C 180,E1 2148.501,E2 2148.501} C_VEL
LIN {X 0,Y 570.926,Z 831.81,A -85,B 0,C 180,E1 2156.188,E2 2156.188} C_VEL
LIN {X 0,Y 570.812,Z 831.81,A -85,B 0,C 180,E1 2163.81,E2 2163.81} C_VEL
LIN {X 0,Y 570.715,Z 831.81,A -85,B 0,C 180,E1 2171.503,E2 2171.503} C_VEL
LIN {X 0,Y 570.605,Z 831.81,A -85,B 0,C 180,E1 2179.417,E2 2179.417} C_VEL
LIN {X 0,Y 570.467,Z 831.81,A -85,B 0,C 180,E1 2186.981,E2 2186.981} C_VEL
LIN {X 0,Y 570.442,Z 831.81,A -85,B 0,C 180,E1 2193.071,E2 2193.071} C_VEL
LIN {X 0,Y 570.705,Z 831.81,A -85,B 0,C 180,E1 2200.726,E2 2200.726} C_VEL
LIN {X 0,Y 570.661,Z 831.81,A -85,B 0,C 180,E1 2209.343,E2 2209.343} C_VEL
LIN {X 0,Y 570.605,Z 831.81,A -85,B 0,C 180,E1 2218.761,E2 2218.761} C_VEL
LIN {X 0,Y 570.457,Z 831.81,A -85,B 0,C 180,E1 2226.607,E2 2226.607} C_VEL
LIN {X 0,Y 570.821,Z 831.81,A -85,B 0,C 180,E1 2235.371,E2 2235.371} C_VEL
LIN {X 0,Y 571.11,Z 831.81,A -85,B 0,C 180,E1 2243.132,E2 2243.132} C_VEL
LIN {X 0,Y 570.548,Z 831.81,A -85,B 0,C 180,E1 2250.762,E2 2250.762} C_VEL
LIN {X 0,Y 571.417,Z 833.479,A -85,B 0,C 180,E1 2257.247,E2 2257.247} C_VEL
LIN {X 0,Y 572.339,Z 874.171,A -85,B 0,C 180,E1 2259.25,E2 2259.25} C_VEL
LIN {X 0,Y 571.947,Z 905.468,A -85,B 0,C 180,E1 2262.449,E2 2262.449} C_VEL
LIN {X 0,Y 571.704,Z 923.437,A -85,B 0,C 180,E1 2266.183,E2 2266.183} C_VEL
LIN {X 0,Y 571.411,Z 928.899,A -85,B 0,C 180,E1 2269.467,E2 2269.467} C_VEL
LIN {X 0,Y 571.745,Z 923.548,A -85,B 0,C 180,E1 2273.69,E2 2273.69} C_VEL
LIN {X 0,Y 571.941,Z 904.037,A -85,B 0,C 180,E1 2277.667,E2 2277.667} C_VEL
LIN {X 0,Y 572.384,Z 872.751,A -85,B 0,C 180,E1 2280.759,E2 2280.759} C_VEL
LIN {X 0,Y 571.2,Z 831.81,A -85,B 0,C 180,E1 2282.839,E2 2282.839} C_VEL
LIN {X 0,Y 570.701,Z 831.81,A -85,B 0,C 180,E1 2290.724,E2 2290.724} C_VEL
LIN {X 0,Y 570.614,Z 831.81,A -85,B 0,C 180,E1 2299.339,E2 2299.339} C_VEL
LIN {X 0,Y 570.6,Z 831.81,A -85,B 0,C 180,E1 2308.76,E2 2308.76} C_VEL
LIN {X 0,Y 570.446,Z 831.81,A -85,B 0,C 180,E1 2316.605,E2 2316.605} C_VEL
LIN {X 0,Y 570.811,Z 831.81,A -85,B 0,C 180,E1 2325.371,E2 2325.371} C_VEL
LIN {X 0,Y 571.119,Z 831.81,A -85,B 0,C 180,E1 2333.134,E2 2333.134} C_VEL
LIN {X 0,Y 570.966,Z 831.81,A -85,B 0,C 180,E1 2340.763,E2 2340.763} C_VEL
LIN {X 0,Y 570.812,Z 831.81,A -85,B 0,C 180,E1 2348.41,E2 2348.41} C_VEL
LIN {X 0,Y 571.066,Z 831.81,A -85,B 0,C 180,E1 2354.354,E2 2354.354} C_VEL
LIN {X 0,Y 562.704,Z 831.81,A -85,B 0,C 180,E1 2357.845,E2 2357.845} C_VEL
LIN {X 0,Y 562.773,Z 831.81,A -85,B 0,C 180,E1 2366.422,E2 2366.422} C_VEL
LIN {X 0,Y 562.821,Z 831.81,A -85,B 0,C 180,E1 2375.434,E2 2375.434} C_VEL
LIN {X 0,Y 562.694,Z 831.81,A -85,B 0,C 180,E1 2385.623,E2 2385.623} C_VEL
LIN {X 0,Y 562.572,Z 831.81,A -85,B 0,C 180,E1 2394.552,E2 2394.552} C_VEL
LIN {X 0,Y 562.781,Z 831.81,A -85,B 0,C 180,E1 2403.582,E2 2403.582} C_VEL
LIN {X 0,Y 563.202,Z 833.501,A -85,B 0,C 180,E1 2407.162,E2 2407.162} C_VEL
LIN {X 0,Y 566.607,Z 856.384,A -85,B 0,C 180,E1 2407.615,E2 2407.615} C_VEL
LIN {X 0,Y 566.495,Z 930.363,A -85,B 0,C 180,E1 2408.998,E2 2408.998} C_VEL
LIN {X 0,Y 565.507,Z 981.011,A -85,B 0,C 180,E1 2411.519,E2 2411.519} C_VEL
LIN {X 0,Y 564.511,Z 1024.289,A -85,B 0,C 180,E1 2415.38,E2 2415.38} C_VEL
LIN {X 0,Y 563.699,Z 1056.692,A -85,B 0,C 180,E1 2420.314,E2 2420.314} C_VEL
LIN {X 0,Y 563.343,Z 1074.38,A -85,B 0,C 180,E1 2425.528,E2 2425.528} C_VEL
LIN {X 0,Y 563.23,Z 1078.838,A -85,B 0,C 180,E1 2430.772,E2 2430.772} C_VEL
LIN {X 0,Y 563.142,Z 1070.117,A -85,B 0,C 180,E1 2436.188,E2 2436.188} C_VEL
LIN {X 0,Y 563.571,Z 1047.723,A -85,B 0,C 180,E1 2441.369,E2 2441.369} C_VEL
LIN {X 0,Y 564.503,Z 1011.489,A -85,B 0,C 180,E1 2445.995,E2 2445.995} C_VEL
LIN {X 0,Y 565.858,Z 964.679,A -85,B 0,C 180,E1 2449.485,E2 2449.485} C_VEL
LIN {X 0,Y 566.871,Z 912.646,A -85,B 0,C 180,E1 2451.505,E2 2451.505} C_VEL
LIN {X 0,Y 564.325,Z 836.062,A -85,B 0,C 180,E1 2452.755,E2 2452.755} C_VEL
LIN {X 0,Y 563.089,Z 831.81,A -85,B 0,C 180,E1 2453.003,E2 2453.003} C_VEL
LIN {X 0,Y 562.346,Z 831.81,A -85,B 0,C 180,E1 2461.774,E2 2461.774} C_VEL
LIN {X 0,Y 562.444,Z 831.81,A -85,B 0,C 180,E1 2469.732,E2 2469.732} C_VEL
LIN {X 0,Y 562.322,Z 831.81,A -85,B 0,C 180,E1 2477.915,E2 2477.915} C_VEL
LIN {X 0,Y 562.362,Z 831.81,A -85,B 0,C 180,E1 2485.391,E2 2485.391} C_VEL
LIN {X 0,Y 562.547,Z 831.81,A -85,B 0,C 180,E1 2493.566,E2 2493.566} C_VEL
LIN {X 0,Y 562.761,Z 831.81,A -85,B 0,C 180,E1 2501.931,E2 2501.931} C_VEL
LIN {X 0,Y 562.77,Z 831.81,A -85,B 0,C 180,E1 2509.903,E2 2509.903} C_VEL
LIN {X 0,Y 562.756,Z 831.81,A -85,B 0,C 180,E1 2517.68,E2 2517.68} C_VEL
LIN {X 0,Y 562.819,Z 831.81,A -85,B 0,C 180,E1 2523.864,E2 2523.864} C_VEL
LIN {X 0,Y 562.708,Z 831.81,A -85,B 0,C 180,E1 2531.669,E2 2531.669} C_VEL
LIN {X 0,Y 562.625,Z 831.81,A -85,B 0,C 180,E1 2539.703,E2 2539.703} C_VEL
LIN {X 0,Y 562.595,Z 831.81,A -85,B 0,C 180,E1 2548.167,E2 2548.167} C_VEL
LIN {X 0,Y 562.497,Z 831.81,A -85,B 0,C 180,E1 2557.375,E2 2557.375} C_VEL
LIN {X 0,Y 562.792,Z 831.81,A -85,B 0,C 180,E1 2566.56,E2 2566.56} C_VEL
LIN {X 0,Y 562.794,Z 831.81,A -85,B 0,C 180,E1 2576.442,E2 2576.442} C_VEL
LIN {X 0,Y 562.814,Z 831.81,A -85,B 0,C 180,E1 2585.296,E2 2585.296} C_VEL
LIN {X 0,Y 562.841,Z 831.81,A -85,B 0,C 180,E1 2595.159,E2 2595.159} C_VEL
LIN {X 0,Y 563.12,Z 831.81,A -85,B 0,C 180,E1 2603.034,E2 2603.034} C_VEL
LIN {X 0,Y 562.561,Z 831.81,A -85,B 0,C 180,E1 2610.773,E2 2610.773} C_VEL
LIN {X 0,Y 563.283,Z 833.483,A -85,B 0,C 180,E1 2617.06,E2 2617.06} C_VEL
LIN {X 0,Y 564.439,Z 872.656,A -85,B 0,C 180,E1 2618.99,E2 2618.99} C_VEL
LIN {X 0,Y 564.012,Z 904.71,A -85,B 0,C 180,E1 2622.233,E2 2622.233} C_VEL
LIN {X 0,Y 563.609,Z 924.292,A -85,B 0,C 180,E1 2626.422,E2 2626.422} C_VEL
LIN {X 0,Y 563.402,Z 928.947,A -85,B 0,C 180,E1 2629.675,E2 2629.675} C_VEL
LIN {X 0,Y 563.701,Z 922.638,A -85,B 0,C 180,E1 2634.049,E2 2634.049} C_VEL
LIN {X 0,Y 563.973,Z 901.711,A -85,B 0,C 180,E1 2638.092,E2 2638.092} C_VEL
LIN {X 0,Y 564.501,Z 868.659,A -85,B 0,C 180,E1 2641.194,E2 2641.194} C_VEL
LIN {X 0,Y 563.115,Z 831.81,A -85,B 0,C 180,E1 2643.016,E2 2643.016} C_VEL
LIN {X 0,Y 562.368,Z 831.81,A -85,B 0,C 180,E1 2652.089,E2 2652.089} C_VEL
LIN {X 0,Y 562.295,Z 831.81,A -85,B 0,C 180,E1 2660.279,E2 2660.279} C_VEL
LIN {X 0,Y 562.618,Z 831.81,A -85,B 0,C 180,E1 2668.266,E2 2668.266} C_VEL
LIN {X 0,Y 562.324,Z 831.81,A -85,B 0,C 180,E1 2676.964,E2 2676.964} C_VEL
LIN {X 0,Y 562.833,Z 831.81,A -85,B 0,C 180,E1 2685.159,E2 2685.159} C_VEL
LIN {X 0,Y 563.129,Z 831.81,A -85,B 0,C 180,E1 2693.036,E2 2693.036} C_VEL
LIN {X 0,Y 562.967,Z 831.81,A -85,B 0,C 180,E1 2700.774,E2 2700.774} C_VEL
LIN {X 0,Y 562.792,Z 831.81,A -85,B 0,C 180,E1 2708.531,E2 2708.531} C_VEL
LIN {X 0,Y 562.609,Z 831.81,A -85,B 0,C 180,E1 2716.455,E2 2716.455} C_VEL
LIN {X 0,Y 562.704,Z 831.81,A -85,B 0,C 180,E1 2717.845,E2 2717.845} C_VEL
LIN {X 0,Y 554.891,Z 831.81,A -85,B 0,C 180,E1 2721.411,E2 2721.411} C_VEL
LIN {X 0,Y 554.524,Z 831.81,A -85,B 0,C 180,E1 2730.454,E2 2730.454} C_VEL
LIN {X 0,Y 554.525,Z 831.81,A -85,B 0,C 180,E1 2738.745,E2 2738.745} C_VEL
LIN {X 0,Y 554.525,Z 831.81,A -85,B 0,C 180,E1 2746.492,E2 2746.492} C_VEL
LIN {X 0,Y 554.608,Z 831.81,A -85,B 0,C 180,E1 2753.965,E2 2753.965} C_VEL
LIN {X 0,Y 554.781,Z 831.81,A -85,B 0,C 180,E1 2763.171,E2 2763.171} C_VEL
LIN {X 0,Y 555.072,Z 833.334,A -85,B 0,C 180,E1 2766.806,E2 2766.806} C_VEL
LIN {X 0,Y 559.165,Z 852.481,A -85,B 0,C 180,E1 2767.247,E2 2767.247} C_VEL
LIN {X 0,Y 559.033,Z 929.374,A -85,B 0,C 180,E1 2768.669,E2 2768.669} C_VEL
LIN {X 0,Y 557.859,Z 981.013,A -85,B 0,C 180,E1 2771.257,E2 2771.257} C_VEL
LIN {X 0,Y 556.693,Z 1024.225,A -85,B 0,C 180,E1 2775.162,E2 2775.162} C_VEL
LIN {X 0,Y 555.762,Z 1056.691,A -85,B 0,C 180,E1 2780.174,E2 2780.174} C_VEL
LIN {X 0,Y 555.452,Z 1074.049,A -85,B 0,C 180,E1 2785.299,E2 2785.299} C_VEL
LIN {X 0,Y 555.226,Z 1078.838,A -85,B 0,C 180,E1 2790.783,E2 2790.783} C_VEL
LIN {X 0,Y 555.135,Z 1070.118,A -85,B 0,C 180,E1 2796.278,E2 2796.278} C_VEL
LIN {X 0,Y 555.628,Z 1048.901,A -85,B 0,C 180,E1 2801.326,E2 2801.326} C_VEL
LIN {X 0,Y 556.696,Z 1013.478,A -85,B 0,C 180,E1 2806.022,E2 2806.022} C_VEL
LIN {X 0,Y 558.199,Z 968.176,A -85,B 0,C 180,E1 2809.557,E2 2809.557} C_VEL
LIN {X 0,Y 559.4,Z 916.14,A -85,B 0,C 180,E1 2811.714,E2 2811.714} C_VEL
LIN {X 0,Y 557.302,Z 839.082,A -85,B 0,C 180,E1 2813.017,E2 2813.017} C_VEL
LIN {X 0,Y 554.996,Z 831.81,A -85,B 0,C 180,E1 2813.358,E2 2813.358} C_VEL
LIN {X 0,Y 554.334,Z 831.81,A -85,B 0,C 180,E1 2822.265,E2 2822.265} C_VEL
LIN {X 0,Y 554.417,Z 831.81,A -85,B 0,C 180,E1 2830.034,E2 2830.034} C_VEL
LIN {X 0,Y 554.344,Z 831.81,A -85,B 0,C 180,E1 2837.874,E2 2837.874} C_VEL
LIN {X 0,Y 554.269,Z 831.81,A -85,B 0,C 180,E1 2845.852,E2 2845.852} C_VEL
LIN {X 0,Y 554.571,Z 831.81,A -85,B 0,C 180,E1 2853.156,E2 2853.156} C_VEL
LIN {X 0,Y 554.78,Z 831.81,A -85,B 0,C 180,E1 2861.662,E2 2861.662} C_VEL
LIN {X 0,Y 554.788,Z 831.81,A -85,B 0,C 180,E1 2869.756,E2 2869.756} C_VEL
LIN {X 0,Y 554.756,Z 831.81,A -85,B 0,C 180,E1 2877.647,E2 2877.647} C_VEL
LIN {X 0,Y 554.835,Z 831.81,A -85,B 0,C 180,E1 2883.919,E2 2883.919} C_VEL
LIN {X 0,Y 554.706,Z 831.81,A -85,B 0,C 180,E1 2891.839,E2 2891.839} C_VEL
LIN {X 0,Y 554.659,Z 831.81,A -85,B 0,C 180,E1 2899.998,E2 2899.998} C_VEL
LIN {X 0,Y 554.689,Z 831.81,A -85,B 0,C 180,E1 2908.605,E2 2908.605} C_VEL
LIN {X 0,Y 554.606,Z 831.81,A -85,B 0,C 180,E1 2918.755,E2 2918.755} C_VEL
LIN {X 0,Y 554.675,Z 831.81,A -85,B 0,C 180,E1 2928.798,E2 2928.798} C_VEL
LIN {X 0,Y 554.65,Z 831.81,A -85,B 0,C 180,E1 2937.756,E2 2937.756} C_VEL
LIN {X 0,Y 554.398,Z 831.81,A -85,B 0,C 180,E1 2946.615,E2 2946.615} C_VEL
LIN {X 0,Y 554.845,Z 831.81,A -85,B 0,C 180,E1 2954.94,E2 2954.94} C_VEL
LIN {X 0,Y 555.134,Z 831.81,A -85,B 0,C 180,E1 2962.934,E2 2962.934} C_VEL
LIN {X 0,Y 554.549,Z 831.81,A -85,B 0,C 180,E1 2970.784,E2 2970.784} C_VEL
LIN {X 0,Y 555.149,Z 833.495,A -85,B 0,C 180,E1 2976.868,E2 2976.868} C_VEL
LIN {X 0,Y 556.572,Z 872.498,A -85,B 0,C 180,E1 2978.822,E2 2978.822} C_VEL
LIN {X 0,Y 556.073,Z 903.955,A -85,B 0,C 180,E1 2982.01,E2 2982.01} C_VEL
LIN {X 0,Y 555.755,Z 922.766,A -85,B 0,C 180,E1 2985.846,E2 2985.846} C_VEL
LIN {X 0,Y 555.37,Z 929,A -85,B 0,C 180,E1 2989.972,E2 2989.972} C_VEL
LIN {X 0,Y 555.636,Z 921.692,A -85,B 0,C 180,E1 2994.392,E2 2994.392} C_VEL
LIN {X 0,Y 555.972,Z 900.344,A -85,B 0,C 180,E1 2998.394,E2 2998.394} C_VEL
LIN {X 0,Y 556.629,Z 866.441,A -85,B 0,C 180,E1 3001.499,E2 3001.499} C_VEL
LIN {X 0,Y 555.007,Z 831.81,A -85,B 0,C 180,E1 3003.263,E2 3003.263} C_VEL
LIN {X 0,Y 554.373,Z 831.81,A -85,B 0,C 180,E1 3012.118,E2 3012.118} C_VEL
LIN {X 0,Y 554.349,Z 831.81,A -85,B 0,C 180,E1 3019.96,E2 3019.96} C_VEL
LIN {X 0,Y 554.641,Z 831.81,A -85,B 0,C 180,E1 3027.755,E2 3027.755} C_VEL
LIN {X 0,Y 554.384,Z 831.81,A -85,B 0,C 180,E1 3036.615,E2 3036.615} C_VEL
LIN {X 0,Y 554.841,Z 831.81,A -85,B 0,C 180,E1 3044.941,E2 3044.941} C_VEL
LIN {X 0,Y 555.14,Z 831.81,A -85,B 0,C 180,E1 3052.935,E2 3052.935} C_VEL
LIN {X 0,Y 554.962,Z 831.81,A -85,B 0,C 180,E1 3060.785,E2 3060.785} C_VEL
LIN {X 0,Y 554.803,Z 831.81,A -85,B 0,C 180,E1 3068.655,E2 3068.655} C_VEL
LIN {X 0,Y 554.608,Z 831.81,A -85,B 0,C 180,E1 3076.699,E2 3076.699} C_VEL
LIN {X 0,Y 554.891,Z 831.81,A -85,B 0,C 180,E1 3081.411,E2 3081.411} C_VEL
LIN {X 0,Y 546.473,Z 831.81,A -85,B 0,C 180,E1 3085.009,E2 3085.009} C_VEL
LIN {X 0,Y 546.341,Z 831.81,A -85,B 0,C 180,E1 3092.799,E2 3092.799} C_VEL
LIN {X 0,Y 546.43,Z 831.81,A -85,B 0,C 180,E1 3100.746,E2 3100.746} C_VEL
LIN {X 0,Y 546.304,Z 831.81,A -85,B 0,C 180,E1 3109.248,E2 3109.248} C_VEL
LIN {X 0,Y 546.307,Z 831.81,A -85,B 0,C 180,E1 3117.92,E2 3117.92} C_VEL
LIN {X 0,Y 546.907,Z 832.889,A -85,B 0,C 180,E1 3126.433,E2 3126.433} C_VEL
LIN {X 0,Y 551.828,Z 855.608,A -85,B 0,C 180,E1 3126.971,E2 3126.971} C_VEL
LIN {X 0,Y 551.55,Z 929.623,A -85,B 0,C 180,E1 3128.374,E2 3128.374} C_VEL
LIN {X 0,Y 550.177,Z 981.016,A -85,B 0,C 180,E1 3130.985,E2 3130.985} C_VEL
LIN {X 0,Y 548.854,Z 1024.223,A -85,B 0,C 180,E1 3134.945,E2 3134.945} C_VEL
LIN {X 0,Y 547.861,Z 1056.691,A -85,B 0,C 180,E1 3140.031,E2 3140.031} C_VEL
LIN {X 0,Y 547.472,Z 1074.048,A -85,B 0,C 180,E1 3145.23,E2 3145.23} C_VEL
LIN {X 0,Y 547.23,Z 1078.838,A -85,B 0,C 180,E1 3150.795,E2 3150.795} C_VEL
LIN {X 0,Y 547.246,Z 1071.253,A -85,B 0,C 180,E1 3155.969,E2 3155.969} C_VEL
LIN {X 0,Y 547.683,Z 1049.803,A -85,B 0,C 180,E1 3161.326,E2 3161.326} C_VEL
LIN {X 0,Y 548.866,Z 1015.4,A -85,B 0,C 180,E1 3166.051,E2 3166.051} C_VEL
LIN {X 0,Y 550.56,Z 969.881,A -85,B 0,C 180,E1 3169.734,E2 3169.734} C_VEL
LIN {X 0,Y 551.95,Z 917.466,A -85,B 0,C 180,E1 3171.987,E2 3171.987} C_VEL
LIN {X 0,Y 549.855,Z 840.917,A -85,B 0,C 180,E1 3173.321,E2 3173.321} C_VEL
LIN {X 0,Y 546.964,Z 831.81,A -85,B 0,C 180,E1 3173.722,E2 3173.722} C_VEL
LIN {X 0,Y 546.356,Z 831.81,A -85,B 0,C 180,E1 3182.795,E2 3182.795} C_VEL
LIN {X 0,Y 546.425,Z 831.81,A -85,B 0,C 180,E1 3190.742,E2 3190.742} C_VEL
LIN {X 0,Y 546.322,Z 831.81,A -85,B 0,C 180,E1 3199.244,E2 3199.244} C_VEL
LIN {X 0,Y 546.275,Z 831.81,A -85,B 0,C 180,E1 3207.918,E2 3207.918} C_VEL
LIN {X 0,Y 546.337,Z 831.81,A -85,B 0,C 180,E1 3216.246,E2 3216.246} C_VEL
LIN {X 0,Y 546.807,Z 831.81,A -85,B 0,C 180,E1 3224.711,E2 3224.711} C_VEL
LIN {X 0,Y 547.347,Z 831.81,A -85,B 0,C 180,E1 3234.429,E2 3234.429} C_VEL
LIN {X 0,Y 547.217,Z 831.81,A -85,B 0,C 180,E1 3242.383,E2 3242.383} C_VEL
LIN {X 0,Y 546.919,Z 831.81,A -85,B 0,C 180,E1 3250.39,E2 3250.39} C_VEL
LIN {X 0,Y 546.647,Z 831.81,A -85,B 0,C 180,E1 3258.617,E2 3258.617} C_VEL
LIN {X 0,Y 546.501,Z 831.81,A -85,B 0,C 180,E1 3267.27,E2 3267.27} C_VEL
LIN {X 0,Y 546.149,Z 831.81,A -85,B 0,C 180,E1 3274.946,E2 3274.946} C_VEL
LIN {X 0,Y 546.322,Z 831.81,A -85,B 0,C 180,E1 3282.887,E2 3282.887} C_VEL
LIN {X 0,Y 546.435,Z 831.81,A -85,B 0,C 180,E1 3289.795,E2 3289.795} C_VEL
LIN {X 0,Y 546.46,Z 831.81,A -85,B 0,C 180,E1 3299.086,E2 3299.086} C_VEL
LIN {X 0,Y 546.495,Z 831.81,A -85,B 0,C 180,E1 3306.256,E2 3306.256} C_VEL
LIN {X 0,Y 546.845,Z 831.81,A -85,B 0,C 180,E1 3314.714,E2 3314.714} C_VEL
LIN {X 0,Y 547.135,Z 831.81,A -85,B 0,C 180,E1 3322.83,E2 3322.83} C_VEL
LIN {X 0,Y 546.546,Z 831.81,A -85,B 0,C 180,E1 3330.795,E2 3330.795} C_VEL
LIN {X 0,Y 547.058,Z 833.464,A -85,B 0,C 180,E1 3336.67,E2 3336.67} C_VEL
LIN {X 0,Y 548.703,Z 869.558,A -85,B 0,C 180,E1 3338.449,E2 3338.449} C_VEL
LIN {X 0,Y 548.106,Z 901.749,A -85,B 0,C 180,E1 3341.587,E2 3341.587} C_VEL
LIN {X 0,Y 547.773,Z 922.415,A -85,B 0,C 180,E1 3345.671,E2 3345.671} C_VEL
LIN {X 0,Y 547.33,Z 928.939,A -85,B 0,C 180,E1 3350.278,E2 3350.278} C_VEL
LIN {X 0,Y 547.52,Z 920.475,A -85,B 0,C 180,E1 3354.815,E2 3354.815} C_VEL
LIN {X 0,Y 548.013,Z 897.687,A -85,B 0,C 180,E1 3358.854,E2 3358.854} C_VEL
LIN {X 0,Y 548.798,Z 862.54,A -85,B 0,C 180,E1 3361.91,E2 3361.91} C_VEL
LIN {X 0,Y 546.941,Z 831.81,A -85,B 0,C 180,E1 3363.408,E2 3363.408} C_VEL
LIN {X 0,Y 546.3,Z 831.81,A -85,B 0,C 180,E1 3372.888,E2 3372.888} C_VEL
LIN {X 0,Y 546.386,Z 831.81,A -85,B 0,C 180,E1 3379.799,E2 3379.799} C_VEL
LIN {X 0,Y 546.447,Z 831.81,A -85,B 0,C 180,E1 3389.085,E2 3389.085} C_VEL
LIN {X 0,Y 546.482,Z 831.81,A -85,B 0,C 180,E1 3396.256,E2 3396.256} C_VEL
LIN {X 0,Y 546.844,Z 831.81,A -85,B 0,C 180,E1 3404.715,E2 3404.715} C_VEL
LIN {X 0,Y 547.142,Z 831.81,A -85,B 0,C 180,E1 3412.831,E2 3412.831} C_VEL
LIN {X 0,Y 546.973,Z 831.81,A -85,B 0,C 180,E1 3420.796,E2 3420.796} C_VEL
LIN {X 0,Y 546.788,Z 831.81,A -85,B 0,C 180,E1 3428.782,E2 3428.782} C_VEL
LIN {X 0,Y 546.63,Z 831.81,A -85,B 0,C 180,E1 3436.95,E2 3436.95} C_VEL
LIN {X 0,Y 546.473,Z 831.81,A -85,B 0,C 180,E1 3445.009,E2 3445.009} C_VEL
LIN {X 0,Y 538.632,Z 831.81,A -85,B 0,C 180,E1 3448.681,E2 3448.681} C_VEL
LIN {X 0,Y 538.67,Z 831.81,A -85,B 0,C 180,E1 3457.284,E2 3457.284} C_VEL
LIN {X 0,Y 538.432,Z 831.81,A -85,B 0,C 180,E1 3466.329,E2 3466.329} C_VEL
LIN {X 0,Y 538.377,Z 831.81,A -85,B 0,C 180,E1 3474.702,E2 3474.702} C_VEL
LIN {X 0,Y 538.676,Z 831.81,A -85,B 0,C 180,E1 3484.109,E2 3484.109} C_VEL
LIN {X 0,Y 538.918,Z 833.421,A -85,B 0,C 180,E1 3486.07,E2 3486.07} C_VEL
LIN {X 0,Y 544.49,Z 855.487,A -85,B 0,C 180,E1 3486.64,E2 3486.64} C_VEL
LIN {X 0,Y 544.119,Z 929.045,A -85,B 0,C 180,E1 3488.043,E2 3488.043} C_VEL
LIN {X 0,Y 542.522,Z 981.018,A -85,B 0,C 180,E1 3490.706,E2 3490.706} C_VEL
LIN {X 0,Y 541.039,Z 1024.06,A -85,B 0,C 180,E1 3494.703,E2 3494.703} C_VEL
LIN {X 0,Y 539.934,Z 1056.69,A -85,B 0,C 180,E1 3499.883,E2 3499.883} C_VEL
LIN {X 0,Y 539.509,Z 1074.048,A -85,B 0,C 180,E1 3505.16,E2 3505.16} C_VEL
LIN {X 0,Y 539.226,Z 1078.837,A -85,B 0,C 180,E1 3510.807,E2 3510.807} C_VEL
LIN {X 0,Y 539.228,Z 1071.253,A -85,B 0,C 180,E1 3516.058,E2 3516.058} C_VEL
LIN {X 0,Y 539.688,Z 1049.476,A -85,B 0,C 180,E1 3521.558,E2 3521.558} C_VEL
LIN {X 0,Y 541.029,Z 1015.399,A -85,B 0,C 180,E1 3526.29,E2 3526.29} C_VEL
LIN {X 0,Y 542.933,Z 969.879,A -85,B 0,C 180,E1 3530.023,E2 3530.023} C_VEL
LIN {X 0,Y 544.531,Z 917.465,A -85,B 0,C 180,E1 3532.302,E2 3532.302} C_VEL
LIN {X 0,Y 542.47,Z 842.615,A -85,B 0,C 180,E1 3533.634,E2 3533.634} C_VEL
LIN {X 0,Y 538.903,Z 831.81,A -85,B 0,C 180,E1 3534.099,E2 3534.099} C_VEL
LIN {X 0,Y 538.402,Z 831.81,A -85,B 0,C 180,E1 3543.74,E2 3543.74} C_VEL
LIN {X 0,Y 538.447,Z 831.81,A -85,B 0,C 180,E1 3551.674,E2 3551.674} C_VEL
LIN {X 0,Y 538.478,Z 831.81,A -85,B 0,C 180,E1 3560.806,E2 3560.806} C_VEL
LIN {X 0,Y 538.628,Z 831.81,A -85,B 0,C 180,E1 3570.455,E2 3570.455} C_VEL
LIN {X 0,Y 538.812,Z 831.81,A -85,B 0,C 180,E1 3581.099,E2 3581.099} C_VEL
LIN {X 0,Y 538.804,Z 831.81,A -85,B 0,C 180,E1 3589.449,E2 3589.449} C_VEL
LIN {X 0,Y 538.78,Z 831.81,A -85,B 0,C 180,E1 3597.577,E2 3597.577} C_VEL
LIN {X 0,Y 538.84,Z 831.81,A -85,B 0,C 180,E1 3604.036,E2 3604.036} C_VEL
LIN {X 0,Y 538.712,Z 831.81,A -85,B 0,C 180,E1 3612.196,E2 3612.196} C_VEL
LIN {X 0,Y 538.719,Z 831.81,A -85,B 0,C 180,E1 3620.616,E2 3620.616} C_VEL
LIN {X 0,Y 538.655,Z 831.81,A -85,B 0,C 180,E1 3629.54,E2 3629.54} C_VEL
LIN {X 0,Y 538.584,Z 831.81,A -85,B 0,C 180,E1 3639.344,E2 3639.344} C_VEL
LIN {X 0,Y 538.562,Z 831.81,A -85,B 0,C 180,E1 3648.534,E2 3648.534} C_VEL
LIN {X 0,Y 538.506,Z 831.81,A -85,B 0,C 180,E1 3658.578,E2 3658.578} C_VEL
LIN {X 0,Y 538.489,Z 831.81,A -85,B 0,C 180,E1 3666.337,E2 3666.337} C_VEL
LIN {X 0,Y 538.84,Z 831.81,A -85,B 0,C 180,E1 3674.481,E2 3674.481} C_VEL
LIN {X 0,Y 539.132,Z 831.81,A -85,B 0,C 180,E1 3682.723,E2 3682.723} C_VEL
LIN {X 0,Y 538.538,Z 831.81,A -85,B 0,C 180,E1 3690.807,E2 3690.807} C_VEL
LIN {X 0,Y 538.906,Z 833.381,A -85,B 0,C 180,E1 3696.463,E2 3696.463} C_VEL
LIN {X 0,Y 540.914,Z 866.323,A -85,B 0,C 180,E1 3698.063,E2 3698.063} C_VEL
LIN {X 0,Y 540.107,Z 899.36,A -85,B 0,C 180,E1 3701.137,E2 3701.137} C_VEL
LIN {X 0,Y 539.681,Z 920.683,A -85,B 0,C 180,E1 3705.084,E2 3705.084} C_VEL
LIN {X 0,Y 539.299,Z 928.909,A -85,B 0,C 180,E1 3709.492,E2 3709.492} C_VEL
LIN {X 0,Y 539.694,Z 923.123,A -85,B 0,C 180,E1 3714.061,E2 3714.061} C_VEL
LIN {X 0,Y 540.073,Z 902.598,A -85,B 0,C 180,E1 3718.331,E2 3718.331} C_VEL
LIN {X 0,Y 540.888,Z 870.138,A -85,B 0,C 180,E1 3721.589,E2 3721.589} C_VEL
LIN {X 0,Y 539.303,Z 834.204,A -85,B 0,C 180,E1 3723.411,E2 3723.411} C_VEL
LIN {X 0,Y 538.832,Z 831.81,A -85,B 0,C 180,E1 3723.814,E2 3723.814} C_VEL
LIN {X 0,Y 538.385,Z 831.81,A -85,B 0,C 180,E1 3731.671,E2 3731.671} C_VEL
LIN {X 0,Y 538.146,Z 831.81,A -85,B 0,C 180,E1 3740.848,E2 3740.848} C_VEL
LIN {X 0,Y 538.413,Z 831.81,A -85,B 0,C 180,E1 3749.277,E2 3749.277} C_VEL
LIN {X 0,Y 538.147,Z 831.81,A -85,B 0,C 180,E1 3757.624,E2 3757.624} C_VEL
LIN {X 0,Y 538.555,Z 831.81,A -85,B 0,C 180,E1 3766.442,E2 3766.442} C_VEL
LIN {X 0,Y 538.889,Z 831.81,A -85,B 0,C 180,E1 3774.345,E2 3774.345} C_VEL
LIN {X 0,Y 538.869,Z 831.81,A -85,B 0,C 180,E1 3781.335,E2 3781.335} C_VEL
LIN {X 0,Y 538.79,Z 831.81,A -85,B 0,C 180,E1 3788.914,E2 3788.914} C_VEL
LIN {X 0,Y 538.63,Z 831.81,A -85,B 0,C 180,E1 3797.21,E2 3797.21} C_VEL
LIN {X 0,Y 538.592,Z 831.81,A -85,B 0,C 180,E1 3805.899,E2 3805.899} C_VEL
LIN {X 0,Y 538.632,Z 831.81,A -85,B 0,C 180,E1 3808.681,E2 3808.681} C_VEL
LIN {X 0,Y 530.291,Z 831.81,A -85,B 0,C 180,E1 3812.369,E2 3812.369} C_VEL
LIN {X 0,Y 530.371,Z 831.81,A -85,B 0,C 180,E1 3820.691,E2 3820.691} C_VEL
LIN {X 0,Y 530.3,Z 831.81,A -85,B 0,C 180,E1 3829.919,E2 3829.919} C_VEL
LIN {X 0,Y 530.275,Z 831.81,A -85,B 0,C 180,E1 3838.033,E2 3838.033} C_VEL
LIN {X 0,Y 530.865,Z 833.29,A -85,B 0,C 180,E1 3845.682,E2 3845.682} C_VEL
LIN {X 0,Y 537.16,Z 857.447,A -85,B 0,C 180,E1 3846.33,E2 3846.33} C_VEL
LIN {X 0,Y 536.645,Z 930.558,A -85,B 0,C 180,E1 3847.777,E2 3847.777} C_VEL
LIN {X 0,Y 534.862,Z 982.5,A -85,B 0,C 180,E1 3850.526,E2 3850.526} C_VEL
LIN {X 0,Y 533.189,Z 1024.985,A -85,B 0,C 180,E1 3854.584,E2 3854.584} C_VEL
LIN {X 0,Y 531.987,Z 1057.07,A -85,B 0,C 180,E1 3859.811,E2 3859.811} C_VEL
LIN {X 0,Y 531.534,Z 1074.047,A -85,B 0,C 180,E1 3865.087,E2 3865.087} C_VEL
LIN {X 0,Y 531.239,Z 1078.837,A -85,B 0,C 180,E1 3870.819,E2 3870.819} C_VEL
LIN {X 0,Y 531.222,Z 1071.253,A -85,B 0,C 180,E1 3876.15,E2 3876.15} C_VEL
LIN {X 0,Y 531.75,Z 1050.567,A -85,B 0,C 180,E1 3881.524,E2 3881.524} C_VEL
LIN {X 0,Y 533.218,Z 1017.321,A -85,B 0,C 180,E1 3886.323,E2 3886.323} C_VEL
LIN {X 0,Y 535.326,Z 971.747,A -85,B 0,C 180,E1 3890.202,E2 3890.202} C_VEL
LIN {X 0,Y 537.08,Z 919.602,A -85,B 0,C 180,E1 3892.57,E2 3892.57} C_VEL
LIN {X 0,Y 535.255,Z 844.794,A -85,B 0,C 180,E1 3893.941,E2 3893.941} C_VEL
LIN {X 0,Y 530.847,Z 831.81,A -85,B 0,C 180,E1 3894.489,E2 3894.489} C_VEL
LIN {X 0,Y 530.416,Z 831.81,A -85,B 0,C 180,E1 3903.911,E2 3903.911} C_VEL
LIN {X 0,Y 530.494,Z 831.81,A -85,B 0,C 180,E1 3913.153,E2 3913.153} C_VEL
LIN {X 0,Y 530.51,Z 831.81,A -85,B 0,C 180,E1 3922.042,E2 3922.042} C_VEL
LIN {X 0,Y 530.605,Z 831.81,A -85,B 0,C 180,E1 3931.838,E2 3931.838} C_VEL
LIN {X 0,Y 530.842,Z 831.81,A -85,B 0,C 180,E1 3940.804,E2 3940.804} C_VEL
LIN {X 0,Y 530.832,Z 831.81,A -85,B 0,C 180,E1 3949.289,E2 3949.289} C_VEL
LIN {X 0,Y 530.781,Z 831.81,A -85,B 0,C 180,E1 3957.54,E2 3957.54} C_VEL
LIN {X 0,Y 530.834,Z 831.81,A -85,B 0,C 180,E1 3964.097,E2 3964.097} C_VEL
LIN {X 0,Y 530.73,Z 831.81,A -85,B 0,C 180,E1 3972.382,E2 3972.382} C_VEL
LIN {X 0,Y 530.777,Z 831.81,A -85,B 0,C 180,E1 3981.688,E2 3981.688} C_VEL
LIN {X 0,Y 530.531,Z 831.81,A -85,B 0,C 180,E1 3991.95,E2 3991.95} C_VEL
LIN {X 0,Y 530.401,Z 831.81,A -85,B 0,C 180,E1 4000.694,E2 4000.694} C_VEL
LIN {X 0,Y 530.278,Z 831.81,A -85,B 0,C 180,E1 4009.916,E2 4009.916} C_VEL
LIN {X 0,Y 530.465,Z 831.81,A -85,B 0,C 180,E1 4018.045,E2 4018.045} C_VEL
LIN {X 0,Y 530.225,Z 831.81,A -85,B 0,C 180,E1 4027.27,E2 4027.27} C_VEL
LIN {X 0,Y 530.596,Z 831.81,A -85,B 0,C 180,E1 4035.93,E2 4035.93} C_VEL
LIN {X 0,Y 530.855,Z 831.81,A -85,B 0,C 180,E1 4044.257,E2 4044.257} C_VEL
LIN {X 0,Y 530.525,Z 831.81,A -85,B 0,C 180,E1 4050.819,E2 4050.819} C_VEL
LIN {X 0,Y 530.831,Z 833.479,A -85,B 0,C 180,E1 4056.257,E2 4056.257} C_VEL
LIN {X 0,Y 533.14,Z 862.925,A -85,B 0,C 180,E1 4057.667,E2 4057.667} C_VEL
LIN {X 0,Y 532.178,Z 896.847,A -85,B 0,C 180,E1 4060.681,E2 4060.681} C_VEL
LIN {X 0,Y 531.652,Z 920.241,A -85,B 0,C 180,E1 4064.886,E2 4064.886} C_VEL
LIN {X 0,Y 531.297,Z 928.785,A -85,B 0,C 180,E1 4069.176,E2 4069.176} C_VEL
LIN {X 0,Y 531.701,Z 923.607,A -85,B 0,C 180,E1 4073.951,E2 4073.951} C_VEL
LIN {X 0,Y 532.137,Z 904.43,A -85,B 0,C 180,E1 4078.187,E2 4078.187} C_VEL
LIN {X 0,Y 532.952,Z 872.823,A -85,B 0,C 180,E1 4081.564,E2 4081.564} C_VEL
LIN {X 0,Y 531.602,Z 835.903,A -85,B 0,C 180,E1 4083.555,E2 4083.555} C_VEL
LIN {X 0,Y 530.822,Z 831.81,A -85,B 0,C 180,E1 4083.881,E2 4083.881} C_VEL
LIN {X 0,Y 530.247,Z 831.81,A -85,B 0,C 180,E1 4093.129,E2 4093.129} C_VEL
LIN {X 0,Y 530.016,Z 831.81,A -85,B 0,C 180,E1 4102.005,E2 4102.005} C_VEL
LIN {X 0,Y 530.36,Z 831.81,A -85,B 0,C 180,E1 4110.774,E2 4110.774} C_VEL
LIN {X 0,Y 530.005,Z 831.81,A -85,B 0,C 180,E1 4119.029,E2 4119.029} C_VEL
LIN {X 0,Y 530.59,Z 831.81,A -85,B 0,C 180,E1 4125.931,E2 4125.931} C_VEL
LIN {X 0,Y 530.892,Z 831.81,A -85,B 0,C 180,E1 4134.259,E2 4134.259} C_VEL
LIN {X 0,Y 530.996,Z 831.81,A -85,B 0,C 180,E1 4140.82,E2 4140.82} C_VEL
LIN {X 0,Y 530.759,Z 831.81,A -85,B 0,C 180,E1 4149.455,E2 4149.455} C_VEL
LIN {X 0,Y 530.636,Z 831.81,A -85,B 0,C 180,E1 4157.477,E2 4157.477} C_VEL
LIN {X 0,Y 530.623,Z 831.81,A -85,B 0,C 180,E1 4166.317,E2 4166.317} C_VEL
LIN {X 0,Y 530.291,Z 831.81,A -85,B 0,C 180,E1 4172.369,E2 4172.369} C_VEL
LIN {X 0,Y 522.449,Z 831.81,A -85,B 0,C 180,E1 4176.146,E2 4176.146} C_VEL
LIN {X 0,Y 522.479,Z 831.81,A -85,B 0,C 180,E1 4185.371,E2 4185.371} C_VEL
LIN {X 0,Y 522.259,Z 831.81,A -85,B 0,C 180,E1 4195.486,E2 4195.486} C_VEL
LIN {X 0,Y 522.67,Z 831.81,A -85,B 0,C 180,E1 4205.24,E2 4205.24} C_VEL
LIN {X 0,Y 529.848,Z 858.163,A -85,B 0,C 180,E1 4205.994,E2 4205.994} C_VEL
LIN {X 0,Y 529.244,Z 930.558,A -85,B 0,C 180,E1 4207.449,E2 4207.449} C_VEL
LIN {X 0,Y 527.295,Z 981.554,A -85,B 0,C 180,E1 4210.164,E2 4210.164} C_VEL
LIN {X 0,Y 525.393,Z 1024.495,A -85,B 0,C 180,E1 4214.289,E2 4214.289} C_VEL
LIN {X 0,Y 524.13,Z 1055.991,A -85,B 0,C 180,E1 4219.424,E2 4219.424} C_VEL
LIN {X 0,Y 523.577,Z 1074.047,A -85,B 0,C 180,E1 4225.012,E2 4225.012} C_VEL
LIN {X 0,Y 523.252,Z 1078.837,A -85,B 0,C 180,E1 4230.831,E2 4230.831} C_VEL
LIN {X 0,Y 523.238,Z 1071.253,A -85,B 0,C 180,E1 4236.244,E2 4236.244} C_VEL
LIN {X 0,Y 523.786,Z 1050.566,A -85,B 0,C 180,E1 4241.701,E2 4241.701} C_VEL
LIN {X 0,Y 525.372,Z 1017.32,A -85,B 0,C 180,E1 4246.573,E2 4246.573} C_VEL
LIN {X 0,Y 527.719,Z 972.424,A -85,B 0,C 180,E1 4250.462,E2 4250.462} C_VEL
LIN {X 0,Y 529.68,Z 919.603,A -85,B 0,C 180,E1 4252.903,E2 4252.903} C_VEL
LIN {X 0,Y 527.693,Z 846.17,A -85,B 0,C 180,E1 4254.268,E2 4254.268} C_VEL
LIN {X 0,Y 522.821,Z 831.81,A -85,B 0,C 180,E1 4254.89,E2 4254.89} C_VEL
LIN {X 0,Y 522.457,Z 831.81,A -85,B 0,C 180,E1 4264.5,E2 4264.5} C_VEL
LIN {X 0,Y 522.527,Z 831.81,A -85,B 0,C 180,E1 4274.634,E2 4274.634} C_VEL
LIN {X 0,Y 522.391,Z 831.81,A -85,B 0,C 180,E1 4283.445,E2 4283.445} C_VEL
LIN {X 0,Y 522.412,Z 831.81,A -85,B 0,C 180,E1 4293.236,E2 4293.236} C_VEL
LIN {X 0,Y 522.645,Z 831.81,A -85,B 0,C 180,E1 4302.246,E2 4302.246} C_VEL
LIN {X 0,Y 522.759,Z 831.81,A -85,B 0,C 180,E1 4310.81,E2 4310.81} C_VEL
LIN {X 0,Y 523.007,Z 831.81,A -85,B 0,C 180,E1 4319.167,E2 4319.167} C_VEL
LIN {X 0,Y 523.203,Z 831.81,A -85,B 0,C 180,E1 4329.178,E2 4329.178} C_VEL
LIN {X 0,Y 522.777,Z 831.81,A -85,B 0,C 180,E1 4337.745,E2 4337.745} C_VEL
LIN {X 0,Y 522.466,Z 831.81,A -85,B 0,C 180,E1 4346.757,E2 4346.757} C_VEL
LIN {X 0,Y 522.175,Z 831.81,A -85,B 0,C 180,E1 4354.521,E2 4354.521} C_VEL
LIN {X 0,Y 522.262,Z 831.81,A -85,B 0,C 180,E1 4363.067,E2 4363.067} C_VEL
LIN {X 0,Y 522.09,Z 831.81,A -85,B 0,C 180,E1 4371.322,E2 4371.322} C_VEL
LIN {X 0,Y 522.338,Z 831.81,A -85,B 0,C 180,E1 4379.441,E2 4379.441} C_VEL
LIN {X 0,Y 522.248,Z 831.81,A -85,B 0,C 180,E1 4386.903,E2 4386.903} C_VEL
LIN {X 0,Y 522.613,Z 831.81,A -85,B 0,C 180,E1 4395.71,E2 4395.71} C_VEL
LIN {X 0,Y 522.879,Z 831.81,A -85,B 0,C 180,E1 4404.17,E2 4404.17} C_VEL
LIN {X 0,Y 522.513,Z 831.81,A -85,B 0,C 180,E1 4410.832,E2 4410.832} C_VEL
LIN {X 0,Y 522.734,Z 833.537,A -85,B 0,C 180,E1 4415.988,E2 4415.988} C_VEL
LIN {X 0,Y 525.322,Z 862.731,A -85,B 0,C 180,E1 4417.469,E2 4417.469} C_VEL
LIN {X 0,Y 524.238,Z 897.693,A -85,B 0,C 180,E1 4420.65,E2 4420.65} C_VEL
LIN {X 0,Y 523.621,Z 919.806,A -85,B 0,C 180,E1 4424.69,E2 4424.69} C_VEL
LIN {X 0,Y 523.281,Z 928.91,A -85,B 0,C 180,E1 4429.481,E2 4429.481} C_VEL
LIN {X 0,Y 523.702,Z 923.352,A -85,B 0,C 180,E1 4434.104,E2 4434.104} C_VEL
LIN {X 0,Y 524.137,Z 902.95,A -85,B 0,C 180,E1 4438.537,E2 4438.537} C_VEL
LIN {X 0,Y 525.129,Z 871.216,A -85,B 0,C 180,E1 4441.861,E2 4441.861} C_VEL
LIN {X 0,Y 523.618,Z 835.85,A -85,B 0,C 180,E1 4443.819,E2 4443.819} C_VEL
LIN {X 0,Y 522.756,Z 831.81,A -85,B 0,C 180,E1 4444.171,E2 4444.171} C_VEL
LIN {X 0,Y 522.248,Z 831.81,A -85,B 0,C 180,E1 4453.067,E2 4453.067} C_VEL
LIN {X 0,Y 522.03,Z 831.81,A -85,B 0,C 180,E1 4461.317,E2 4461.317} C_VEL
LIN {X 0,Y 522.325,Z 831.81,A -85,B 0,C 180,E1 4469.44,E2 4469.44} C_VEL
LIN {X 0,Y 522.233,Z 831.81,A -85,B 0,C 180,E1 4476.903,E2 4476.903} C_VEL
LIN {X 0,Y 522.606,Z 831.81,A -85,B 0,C 180,E1 4485.711,E2 4485.711} C_VEL
LIN {X 0,Y 522.91,Z 831.81,A -85,B 0,C 180,E1 4494.172,E2 4494.172} C_VEL
LIN {X 0,Y 523.001,Z 831.81,A -85,B 0,C 180,E1 4500.833,E2 4500.833} C_VEL
LIN {X 0,Y 522.778,Z 831.81,A -85,B 0,C 180,E1 4509.189,E2 4509.189} C_VEL
LIN {X 0,Y 522.638,Z 831.81,A -85,B 0,C 180,E1 4517.754,E2 4517.754} C_VEL
LIN {X 0,Y 522.625,Z 831.81,A -85,B 0,C 180,E1 4527.672,E2 4527.672} C_VEL
LIN {X 0,Y 522.449,Z 831.81,A -85,B 0,C 180,E1 4536.146,E2 4536.146} C_VEL
LIN {X 0,Y 514.307,Z 831.81,A -85,B 0,C 180,E1 4539.982,E2 4539.982} C_VEL
LIN {X 0,Y 514.235,Z 831.81,A -85,B 0,C 180,E1 4548.816,E2 4548.816} C_VEL
LIN {X 0,Y 514.356,Z 831.81,A -85,B 0,C 180,E1 4558.915,E2 4558.915} C_VEL
LIN {X 0,Y 514.892,Z 833.745,A -85,B 0,C 180,E1 4565.066,E2 4565.066} C_VEL
LIN {X 0,Y 522.37,Z 861.031,A -85,B 0,C 180,E1 4565.743,E2 4565.743} C_VEL
LIN {X 0,Y 521.743,Z 931.422,A -85,B 0,C 180,E1 4567.163,E2 4567.163} C_VEL
LIN {X 0,Y 519.71,Z 981.291,A -85,B 0,C 180,E1 4569.843,E2 4569.843} C_VEL
LIN {X 0,Y 517.57,Z 1024.493,A -85,B 0,C 180,E1 4574.046,E2 4574.046} C_VEL
LIN {X 0,Y 516.18,Z 1056.52,A -85,B 0,C 180,E1 4579.375,E2 4579.375} C_VEL
LIN {X 0,Y 515.588,Z 1074.047,A -85,B 0,C 180,E1 4584.935,E2 4584.935} C_VEL
LIN {X 0,Y 515.248,Z 1078.837,A -85,B 0,C 180,E1 4590.844,E2 4590.844} C_VEL
LIN {X 0,Y 515.255,Z 1071.253,A -85,B 0,C 180,E1 4596.341,E2 4596.341} C_VEL
LIN {X 0,Y 515.854,Z 1050.566,A -85,B 0,C 180,E1 4601.884,E2 4601.884} C_VEL
LIN {X 0,Y 517.609,Z 1015.956,A -85,B 0,C 180,E1 4606.985,E2 4606.985} C_VEL
LIN {X 0,Y 520.22,Z 970.376,A -85,B 0,C 180,E1 4610.905,E2 4610.905} C_VEL
LIN {X 0,Y 522.215,Z 919.429,A -85,B 0,C 180,E1 4613.223,E2 4613.223} C_VEL
LIN {X 0,Y 520.317,Z 848.44,A -85,B 0,C 180,E1 4614.519,E2 4614.519} C_VEL
LIN {X 0,Y 514.797,Z 831.81,A -85,B 0,C 180,E1 4615.124,E2 4615.124} C_VEL
LIN {X 0,Y 514.408,Z 831.81,A -85,B 0,C 180,E1 4625.118,E2 4625.118} C_VEL
LIN {X 0,Y 514.483,Z 831.81,A -85,B 0,C 180,E1 4633.882,E2 4633.882} C_VEL
LIN {X 0,Y 514.262,Z 831.81,A -85,B 0,C 180,E1 4644.243,E2 4644.243} C_VEL
LIN {X 0,Y 514.312,Z 831.81,A -85,B 0,C 180,E1 4654.151,E2 4654.151} C_VEL
LIN {X 0,Y 514.644,Z 831.81,A -85,B 0,C 180,E1 4663.729,E2 4663.729} C_VEL
LIN {X 0,Y 514.998,Z 831.81,A -85,B 0,C 180,E1 4672.378,E2 4672.378} C_VEL
LIN {X 0,Y 515.182,Z 831.81,A -85,B 0,C 180,E1 4682.531,E2 4682.531} C_VEL
LIN {X 0,Y 514.807,Z 831.81,A -85,B 0,C 180,E1 4691.045,E2 4691.045} C_VEL
LIN {X 0,Y 514.589,Z 831.81,A -85,B 0,C 180,E1 4699.824,E2 4699.824} C_VEL
LIN {X 0,Y 514.47,Z 831.81,A -85,B 0,C 180,E1 4709.522,E2 4709.522} C_VEL
LIN {X 0,Y 514.353,Z 831.81,A -85,B 0,C 180,E1 4719.371,E2 4719.371} C_VEL
LIN {X 0,Y 514.408,Z 831.81,A -85,B 0,C 180,E1 4728.789,E2 4728.789} C_VEL
LIN {X 0,Y 514.35,Z 831.81,A -85,B 0,C 180,E1 4738.914,E2 4738.914} C_VEL
LIN {X 0,Y 514.302,Z 831.81,A -85,B 0,C 180,E1 4746.525,E2 4746.525} C_VEL
LIN {X 0,Y 514.61,Z 831.81,A -85,B 0,C 180,E1 4755.483,E2 4755.483} C_VEL
LIN {X 0,Y 514.881,Z 831.81,A -85,B 0,C 180,E1 4764.079,E2 4764.079} C_VEL
LIN {X 0,Y 514.501,Z 831.81,A -85,B 0,C 180,E1 4770.845,E2 4770.845} C_VEL
LIN {X 0,Y 514.525,Z 833.217,A -85,B 0,C 180,E1 4775.659,E2 4775.659} C_VEL
LIN {X 0,Y 517.76,Z 862.345,A -85,B 0,C 180,E1 4777.155,E2 4777.155} C_VEL
LIN {X 0,Y 516.368,Z 896.621,A -85,B 0,C 180,E1 4780.278,E2 4780.278} C_VEL
LIN {X 0,Y 515.614,Z 919.379,A -85,B 0,C 180,E1 4784.487,E2 4784.487} C_VEL
LIN {X 0,Y 515.326,Z 927.823,A -85,B 0,C 180,E1 4788.011,E2 4788.011} C_VEL
LIN {X 0,Y 515.473,Z 926.758,A -85,B 0,C 180,E1 4792.631,E2 4792.631} C_VEL
LIN {X 0,Y 516.074,Z 910.67,A -85,B 0,C 180,E1 4797.432,E2 4797.432} C_VEL
LIN {X 0,Y 517.099,Z 882.845,A -85,B 0,C 180,E1 4801.163,E2 4801.163} C_VEL
LIN {X 0,Y 517.724,Z 845.602,A -85,B 0,C 180,E1 4803.673,E2 4803.673} C_VEL
LIN {X 0,Y 514.709,Z 831.81,A -85,B 0,C 180,E1 4804.38,E2 4804.38} C_VEL
LIN {X 0,Y 514.241,Z 831.81,A -85,B 0,C 180,E1 4813.907,E2 4813.907} C_VEL
LIN {X 0,Y 514.033,Z 831.81,A -85,B 0,C 180,E1 4822.756,E2 4822.756} C_VEL
LIN {X 0,Y 514.299,Z 831.81,A -85,B 0,C 180,E1 4830.865,E2 4830.865} C_VEL
LIN {X 0,Y 514.124,Z 831.81,A -85,B 0,C 180,E1 4840.157,E2 4840.157} C_VEL
LIN {X 0,Y 514.567,Z 831.81,A -85,B 0,C 180,E1 4848.949,E2 4848.949} C_VEL
LIN {X 0,Y 515.213,Z 831.81,A -85,B 0,C 180,E1 4857.776,E2 4857.776} C_VEL
LIN {X 0,Y 515.006,Z 831.81,A -85,B 0,C 180,E1 4867.622,E2 4867.622} C_VEL
LIN {X 0,Y 514.606,Z 831.81,A -85,B 0,C 180,E1 4876.585,E2 4876.585} C_VEL
LIN {X 0,Y 514.489,Z 831.81,A -85,B 0,C 180,E1 4885.891,E2 4885.891} C_VEL
LIN {X 0,Y 514.391,Z 831.81,A -85,B 0,C 180,E1 4896.143,E2 4896.143} C_VEL
LIN {X 0,Y 514.307,Z 831.81,A -85,B 0,C 180,E1 4899.982,E2 4899.982} C_VEL
LIN {X 0,Y 506.269,Z 831.81,A -85,B 0,C 180,E1 4903.881,E2 4903.881} C_VEL
LIN {X 0,Y 506.292,Z 831.81,A -85,B 0,C 180,E1 4914.234,E2 4914.234} C_VEL
LIN {X 0,Y 506.597,Z 831.81,A -85,B 0,C 180,E1 4924.475,E2 4924.475} C_VEL
LIN {X 0,Y 514.808,Z 861.489,A -85,B 0,C 180,E1 4925.461,E2 4925.461} C_VEL
LIN {X 0,Y 514.129,Z 930.213,A -85,B 0,C 180,E1 4926.863,E2 4926.863} C_VEL
LIN {X 0,Y 511.973,Z 982.788,A -85,B 0,C 180,E1 4929.679,E2 4929.679} C_VEL
LIN {X 0,Y 509.767,Z 1024.493,A -85,B 0,C 180,E1 4933.795,E2 4933.795} C_VEL
LIN {X 0,Y 508.221,Z 1056.689,A -85,B 0,C 180,E1 4939.244,E2 4939.244} C_VEL
LIN {X 0,Y 507.624,Z 1074.046,A -85,B 0,C 180,E1 4944.855,E2 4944.855} C_VEL
LIN {X 0,Y 507.26,Z 1078.836,A -85,B 0,C 180,E1 4950.857,E2 4950.857} C_VEL
LIN {X 0,Y 507.264,Z 1071.253,A -85,B 0,C 180,E1 4956.442,E2 4956.442} C_VEL
LIN {X 0,Y 507.936,Z 1050.566,A -85,B 0,C 180,E1 4962.072,E2 4962.072} C_VEL
LIN {X 0,Y 509.815,Z 1016.796,A -85,B 0,C 180,E1 4967.155,E2 4967.155} C_VEL
LIN {X 0,Y 512.404,Z 973.714,A -85,B 0,C 180,E1 4970.955,E2 4970.955} C_VEL
LIN {X 0,Y 514.581,Z 920.482,A -85,B 0,C 180,E1 4973.461,E2 4973.461} C_VEL
LIN {X 0,Y 512.643,Z 849.957,A -85,B 0,C 180,E1 4974.8,E2 4974.8} C_VEL
LIN {X 0,Y 506.781,Z 831.81,A -85,B 0,C 180,E1 4975.522,E2 4975.522} C_VEL
LIN {X 0,Y 506.44,Z 831.81,A -85,B 0,C 180,E1 4985.755,E2 4985.755} C_VEL
LIN {X 0,Y 506.337,Z 831.81,A -85,B 0,C 180,E1 4995.22,E2 4995.22} C_VEL
LIN {X 0,Y 506.285,Z 831.81,A -85,B 0,C 180,E1 5004.228,E2 5004.228} C_VEL
LIN {X 0,Y 506.313,Z 831.81,A -85,B 0,C 180,E1 5014.237,E2 5014.237} C_VEL
LIN {X 0,Y 506.622,Z 831.81,A -85,B 0,C 180,E1 5023.464,E2 5023.464} C_VEL
LIN {X 0,Y 506.965,Z 831.81,A -85,B 0,C 180,E1 5032.256,E2 5032.256} C_VEL
LIN {X 0,Y 507.181,Z 831.81,A -85,B 0,C 180,E1 5042.571,E2 5042.571} C_VEL
LIN {X 0,Y 506.781,Z 831.81,A -85,B 0,C 180,E1 5051.223,E2 5051.223} C_VEL
LIN {X 0,Y 506.601,Z 831.81,A -85,B 0,C 180,E1 5060.15,E2 5060.15} C_VEL
LIN {X 0,Y 506.481,Z 831.81,A -85,B 0,C 180,E1 5069.629,E2 5069.629} C_VEL
LIN {X 0,Y 506.292,Z 831.81,A -85,B 0,C 180,E1 5080.152,E2 5080.152} C_VEL
LIN {X 0,Y 506.22,Z 831.81,A -85,B 0,C 180,E1 5089.87,E2 5089.87} C_VEL
LIN {X 0,Y 506.336,Z 831.81,A -85,B 0,C 180,E1 5098.671,E2 5098.671} C_VEL
LIN {X 0,Y 506.056,Z 831.81,A -85,B 0,C 180,E1 5107.985,E2 5107.985} C_VEL
LIN {X 0,Y 506.446,Z 831.81,A -85,B 0,C 180,E1 5117.012,E2 5117.012} C_VEL
LIN {X 0,Y 506.834,Z 831.81,A -85,B 0,C 180,E1 5125.707,E2 5125.707} C_VEL
LIN {X 0,Y 506.062,Z 831.81,A -85,B 0,C 180,E1 5132.578,E2 5132.578} C_VEL
LIN {X 0,Y 506.343,Z 832.732,A -85,B 0,C 180,E1 5135.32,E2 5135.32} C_VEL
LIN {X 0,Y 510.157,Z 862.045,A -85,B 0,C 180,E1 5136.833,E2 5136.833} C_VEL
LIN {X 0,Y 508.623,Z 897.258,A -85,B 0,C 180,E1 5140.041,E2 5140.041} C_VEL
LIN {X 0,Y 507.741,Z 919.718,A -85,B 0,C 180,E1 5144.15,E2 5144.15} C_VEL
LIN {X 0,Y 507.364,Z 929.101,A -85,B 0,C 180,E1 5148.304,E2 5148.304} C_VEL
LIN {X 0,Y 507.585,Z 927.406,A -85,B 0,C 180,E1 5152.871,E2 5152.871} C_VEL
LIN {X 0,Y 508.259,Z 911.88,A -85,B 0,C 180,E1 5157.567,E2 5157.567} C_VEL
LIN {X 0,Y 509.437,Z 883.512,A -85,B 0,C 180,E1 5161.419,E2 5161.419} C_VEL
LIN {X 0,Y 509.681,Z 844.82,A -85,B 0,C 180,E1 5164.039,E2 5164.039} C_VEL
LIN {X 0,Y 506.624,Z 831.81,A -85,B 0,C 180,E1 5164.799,E2 5164.799} C_VEL
LIN {X 0,Y 506.205,Z 831.81,A -85,B 0,C 180,E1 5174.789,E2 5174.789} C_VEL
LIN {X 0,Y 506.163,Z 831.81,A -85,B 0,C 180,E1 5184.223,E2 5184.223} C_VEL
LIN {X 0,Y 506.497,Z 831.81,A -85,B 0,C 180,E1 5194.25,E2 5194.25} C_VEL
LIN {X 0,Y 506.62,Z 831.81,A -85,B 0,C 180,E1 5205.25,E2 5205.25} C_VEL
LIN {X 0,Y 506.91,Z 831.81,A -85,B 0,C 180,E1 5213.987,E2 5213.987} C_VEL
LIN {X 0,Y 506.995,Z 831.81,A -85,B 0,C 180,E1 5220.859,E2 5220.859} C_VEL
LIN {X 0,Y 506.773,Z 831.81,A -85,B 0,C 180,E1 5229.482,E2 5229.482} C_VEL
LIN {X 0,Y 506.704,Z 831.81,A -85,B 0,C 180,E1 5239.37,E2 5239.37} C_VEL
LIN {X 0,Y 506.464,Z 831.81,A -85,B 0,C 180,E1 5249.634,E2 5249.634} C_VEL
LIN {X 0,Y 506.402,Z 831.81,A -85,B 0,C 180,E1 5257.908,E2 5257.908} C_VEL
LIN {X 0,Y 506.269,Z 831.81,A -85,B 0,C 180,E1 5263.881,E2 5263.881} C_VEL
LIN {X 0,Y 498.129,Z 831.81,A -85,B 0,C 180,E1 5267.835,E2 5267.835} C_VEL
LIN {X 0,Y 498.181,Z 831.81,A -85,B 0,C 180,E1 5277.787,E2 5277.787} C_VEL
LIN {X 0,Y 498.63,Z 832.074,A -85,B 0,C 180,E1 5284.379,E2 5284.379} C_VEL
LIN {X 0,Y 507.295,Z 863.95,A -85,B 0,C 180,E1 5285.201,E2 5285.201} C_VEL
LIN {X 0,Y 506.468,Z 930.452,A -85,B 0,C 180,E1 5286.609,E2 5286.609} C_VEL
LIN {X 0,Y 504.15,Z 982.573,A -85,B 0,C 180,E1 5289.474,E2 5289.474} C_VEL
LIN {X 0,Y 501.863,Z 1026.078,A -85,B 0,C 180,E1 5293.758,E2 5293.758} C_VEL
LIN {X 0,Y 500.271,Z 1056.688,A -85,B 0,C 180,E1 5299.071,E2 5299.071} C_VEL
LIN {X 0,Y 499.651,Z 1074.046,A -85,B 0,C 180,E1 5304.773,E2 5304.773} C_VEL
LIN {X 0,Y 499.256,Z 1078.836,A -85,B 0,C 180,E1 5310.871,E2 5310.871} C_VEL
LIN {X 0,Y 499.251,Z 1071.253,A -85,B 0,C 180,E1 5316.545,E2 5316.545} C_VEL
LIN {X 0,Y 500.002,Z 1050.565,A -85,B 0,C 180,E1 5322.267,E2 5322.267} C_VEL
LIN {X 0,Y 501.947,Z 1017.701,A -85,B 0,C 180,E1 5327.266,E2 5327.266} C_VEL
LIN {X 0,Y 504.694,Z 971.908,A -85,B 0,C 180,E1 5331.29,E2 5331.29} C_VEL
LIN {X 0,Y 506.997,Z 919.361,A -85,B 0,C 180,E1 5333.775,E2 5333.775} C_VEL
LIN {X 0,Y 505.277,Z 852.214,A -85,B 0,C 180,E1 5335.069,E2 5335.069} C_VEL
LIN {X 0,Y 498.717,Z 831.81,A -85,B 0,C 180,E1 5335.894,E2 5335.894} C_VEL
LIN {X 0,Y 498.397,Z 831.81,A -85,B 0,C 180,E1 5346.424,E2 5346.424} C_VEL
LIN {X 0,Y 498.22,Z 831.81,A -85,B 0,C 180,E1 5356.733,E2 5356.733} C_VEL
LIN {X 0,Y 498.13,Z 831.81,A -85,B 0,C 180,E1 5366.907,E2 5366.907} C_VEL
LIN {X 0,Y 498.277,Z 831.81,A -85,B 0,C 180,E1 5375.719,E2 5375.719} C_VEL
LIN {X 0,Y 498.792,Z 831.81,A -85,B 0,C 180,E1 5385.01,E2 5385.01} C_VEL
LIN {X 0,Y 499.029,Z 831.81,A -85,B 0,C 180,E1 5395.638,E2 5395.638} C_VEL
LIN {X 0,Y 499.163,Z 831.81,A -85,B 0,C 180,E1 5402.612,E2 5402.612} C_VEL
LIN {X 0,Y 498.756,Z 831.81,A -85,B 0,C 180,E1 5411.406,E2 5411.406} C_VEL
LIN {X 0,Y 498.586,Z 831.81,A -85,B 0,C 180,E1 5420.488,E2 5420.488} C_VEL
LIN {X 0,Y 498.461,Z 831.81,A -85,B 0,C 180,E1 5430.155,E2 5430.155} C_VEL
LIN {X 0,Y 498.204,Z 831.81,A -85,B 0,C 180,E1 5440.912,E2 5440.912} C_VEL
LIN {X 0,Y 498.204,Z 831.81,A -85,B 0,C 180,E1 5449.088,E2 5449.088} C_VEL
LIN {X 0,Y 498.27,Z 831.81,A -85,B 0,C 180,E1 5457.792,E2 5457.792} C_VEL
LIN {X 0,Y 498.35,Z 831.81,A -85,B 0,C 180,E1 5465.726,E2 5465.726} C_VEL
LIN {X 0,Y 498.606,Z 831.81,A -85,B 0,C 180,E1 5475.007,E2 5475.007} C_VEL
LIN {X 0,Y 498.882,Z 831.81,A -85,B 0,C 180,E1 5483.888,E2 5483.888} C_VEL
LIN {X 0,Y 498.499,Z 831.81,A -85,B 0,C 180,E1 5490.872,E2 5490.872} C_VEL
LIN {X 0,Y 498.442,Z 833.601,A -85,B 0,C 180,E1 5495.021,E2 5495.021} C_VEL
LIN {X 0,Y 502.573,Z 861.725,A -85,B 0,C 180,E1 5496.501,E2 5496.501} C_VEL
LIN {X 0,Y 500.894,Z 897.395,A -85,B 0,C 180,E1 5499.733,E2 5499.733} C_VEL
LIN {X 0,Y 499.898,Z 920.633,A -85,B 0,C 180,E1 5503.976,E2 5503.976} C_VEL
LIN {X 0,Y 499.47,Z 930.591,A -85,B 0,C 180,E1 5508.603,E2 5508.603} C_VEL
LIN {X 0,Y 499.844,Z 927.066,A -85,B 0,C 180,E1 5513.72,E2 5513.72} C_VEL
LIN {X 0,Y 500.664,Z 909.377,A -85,B 0,C 180,E1 5518.4,E2 5518.4} C_VEL
LIN {X 0,Y 502.036,Z 879.207,A -85,B 0,C 180,E1 5522.141,E2 5522.141} C_VEL
LIN {X 0,Y 501.111,Z 841.437,A -85,B 0,C 180,E1 5524.541,E2 5524.541} C_VEL
LIN {X 0,Y 498.586,Z 831.81,A -85,B 0,C 180,E1 5524.991,E2 5524.991} C_VEL
LIN {X 0,Y 498.148,Z 831.81,A -85,B 0,C 180,E1 5534.282,E2 5534.282} C_VEL
LIN {X 0,Y 498.094,Z 831.81,A -85,B 0,C 180,E1 5543.839,E2 5543.839} C_VEL
LIN {X 0,Y 498.436,Z 831.81,A -85,B 0,C 180,E1 5553.916,E2 5553.916} C_VEL
LIN {X 0,Y 498.602,Z 831.81,A -85,B 0,C 180,E1 5565.008,E2 5565.008} C_VEL
LIN {X 0,Y 498.909,Z 831.81,A -85,B 0,C 180,E1 5573.89,E2 5573.89} C_VEL
LIN {X 0,Y 498.99,Z 831.81,A -85,B 0,C 180,E1 5580.873,E2 5580.873} C_VEL
LIN {X 0,Y 498.769,Z 831.81,A -85,B 0,C 180,E1 5589.636,E2 5589.636} C_VEL
LIN {X 0,Y 498.658,Z 831.81,A -85,B 0,C 180,E1 5598.638,E2 5598.638} C_VEL
LIN {X 0,Y 498.492,Z 831.81,A -85,B 0,C 180,E1 5608.159,E2 5608.159} C_VEL
LIN {X 0,Y 498.287,Z 831.81,A -85,B 0,C 180,E1 5618.638,E2 5618.638} C_VEL
LIN {X 0,Y 498.129,Z 831.81,A -85,B 0,C 180,E1 5627.835,E2 5627.835} C_VEL
LIN {X 0,Y 490.151,Z 831.81,A -85,B 0,C 180,E1 5631.859,E2 5631.859} C_VEL
LIN {X 0,Y 490.559,Z 831.81,A -85,B 0,C 180,E1 5641.852,E2 5641.852} C_VEL
LIN {X 0,Y 490.617,Z 832.533,A -85,B 0,C 180,E1 5644.042,E2 5644.042} C_VEL
LIN {X 0,Y 499.803,Z 866.37,A -85,B 0,C 180,E1 5644.934,E2 5644.934} C_VEL
LIN {X 0,Y 498.823,Z 930.654,A -85,B 0,C 180,E1 5646.347,E2 5646.347} C_VEL
LIN {X 0,Y 496.283,Z 983.105,A -85,B 0,C 180,E1 5649.319,E2 5649.319} C_VEL
LIN {X 0,Y 493.875,Z 1026.371,A -85,B 0,C 180,E1 5653.717,E2 5653.717} C_VEL
LIN {X 0,Y 492.317,Z 1056.67,A -85,B 0,C 180,E1 5658.893,E2 5658.893} C_VEL
LIN {X 0,Y 491.67,Z 1074.045,A -85,B 0,C 180,E1 5664.687,E2 5664.687} C_VEL
LIN {X 0,Y 491.253,Z 1078.836,A -85,B 0,C 180,E1 5670.885,E2 5670.885} C_VEL
LIN {X 0,Y 491.252,Z 1071.252,A -85,B 0,C 180,E1 5676.653,E2 5676.653} C_VEL
LIN {X 0,Y 492.056,Z 1051.456,A -85,B 0,C 180,E1 5682.242,E2 5682.242} C_VEL
LIN {X 0,Y 494.043,Z 1016.962,A -85,B 0,C 180,E1 5687.467,E2 5687.467} C_VEL
LIN {X 0,Y 497.027,Z 970.068,A -85,B 0,C 180,E1 5691.634,E2 5691.634} C_VEL
LIN {X 0,Y 499.517,Z 916.209,A -85,B 0,C 180,E1 5694.154,E2 5694.154} C_VEL
LIN {X 0,Y 497.991,Z 854.749,A -85,B 0,C 180,E1 5695.337,E2 5695.337} C_VEL
LIN {X 0,Y 490.718,Z 831.81,A -85,B 0,C 180,E1 5696.077,E2 5696.077} C_VEL
LIN {X 0,Y 490.318,Z 831.81,A -85,B 0,C 180,E1 5704.93,E2 5704.93} C_VEL
LIN {X 0,Y 490.29,Z 831.81,A -85,B 0,C 180,E1 5714.141,E2 5714.141} C_VEL
LIN {X 0,Y 490.186,Z 831.81,A -85,B 0,C 180,E1 5722.861,E2 5722.861} C_VEL
LIN {X 0,Y 490.263,Z 831.81,A -85,B 0,C 180,E1 5733.328,E2 5733.328} C_VEL
LIN {X 0,Y 490.58,Z 831.81,A -85,B 0,C 180,E1 5742.907,E2 5742.907} C_VEL
LIN {X 0,Y 490.921,Z 831.81,A -85,B 0,C 180,E1 5752.002,E2 5752.002} C_VEL
LIN {X 0,Y 491.164,Z 831.81,A -85,B 0,C 180,E1 5762.655,E2 5762.655} C_VEL
LIN {X 0,Y 490.736,Z 831.81,A -85,B 0,C 180,E1 5771.595,E2 5771.595} C_VEL
LIN {X 0,Y 490.594,Z 831.81,A -85,B 0,C 180,E1 5780.837,E2 5780.837} C_VEL
LIN {X 0,Y 490.349,Z 831.81,A -85,B 0,C 180,E1 5790.707,E2 5790.707} C_VEL
LIN {X 0,Y 490.181,Z 831.81,A -85,B 0,C 180,E1 5800.668,E2 5800.668} C_VEL
LIN {X 0,Y 490.071,Z 831.81,A -85,B 0,C 180,E1 5810.595,E2 5810.595} C_VEL
LIN {X 0,Y 490.219,Z 831.81,A -85,B 0,C 180,E1 5819.284,E2 5819.284} C_VEL
LIN {X 0,Y 490.031,Z 831.81,A -85,B 0,C 180,E1 5829.137,E2 5829.137} C_VEL
LIN {X 0,Y 490.482,Z 831.81,A -85,B 0,C 180,E1 5838.398,E2 5838.398} C_VEL
LIN {X 0,Y 491.177,Z 831.81,A -85,B 0,C 180,E1 5847.343,E2 5847.343} C_VEL
LIN {X 0,Y 490.264,Z 833.158,A -85,B 0,C 180,E1 5854.66,E2 5854.66} C_VEL
LIN {X 0,Y 494.966,Z 863.099,A -85,B 0,C 180,E1 5856.27,E2 5856.27} C_VEL
LIN {X 0,Y 493.166,Z 898.321,A -85,B 0,C 180,E1 5859.52,E2 5859.52} C_VEL
LIN {X 0,Y 492.031,Z 922.065,A -85,B 0,C 180,E1 5863.945,E2 5863.945} C_VEL
LIN {X 0,Y 491.551,Z 931.978,A -85,B 0,C 180,E1 5868.914,E2 5868.914} C_VEL
LIN {X 0,Y 492.022,Z 926.594,A -85,B 0,C 180,E1 5874.51,E2 5874.51} C_VEL
LIN {X 0,Y 492.935,Z 906.404,A -85,B 0,C 180,E1 5879.269,E2 5879.269} C_VEL
LIN {X 0,Y 494.621,Z 873.855,A -85,B 0,C 180,E1 5882.925,E2 5882.925} C_VEL
LIN {X 0,Y 493.15,Z 841.769,A -85,B 0,C 180,E1 5884.878,E2 5884.878} C_VEL
LIN {X 0,Y 490.525,Z 831.81,A -85,B 0,C 180,E1 5885.455,E2 5885.455} C_VEL
LIN {X 0,Y 490.194,Z 831.81,A -85,B 0,C 180,E1 5895.848,E2 5895.848} C_VEL
LIN {X 0,Y 490.179,Z 831.81,A -85,B 0,C 180,E1 5905.125,E2 5905.125} C_VEL
LIN {X 0,Y 490.341,Z 831.81,A -85,B 0,C 180,E1 5915.304,E2 5915.304} C_VEL
LIN {X 0,Y 490.608,Z 831.81,A -85,B 0,C 180,E1 5924.757,E2 5924.757} C_VEL
LIN {X 0,Y 490.92,Z 831.81,A -85,B 0,C 180,E1 5933.79,E2 5933.79} C_VEL
LIN {X 0,Y 491.006,Z 831.81,A -85,B 0,C 180,E1 5940.887,E2 5940.887} C_VEL
LIN {X 0,Y 490.759,Z 831.81,A -85,B 0,C 180,E1 5949.794,E2 5949.794} C_VEL
LIN {X 0,Y 490.607,Z 831.81,A -85,B 0,C 180,E1 5959.367,E2 5959.367} C_VEL
LIN {X 0,Y 490.448,Z 831.81,A -85,B 0,C 180,E1 5968.663,E2 5968.663} C_VEL
LIN {X 0,Y 490.248,Z 831.81,A -85,B 0,C 180,E1 5977.877,E2 5977.877} C_VEL
LIN {X 0,Y 490.136,Z 831.81,A -85,B 0,C 180,E1 5987.838,E2 5987.838} C_VEL
LIN {X 0,Y 490.151,Z 831.81,A -85,B 0,C 180,E1 5991.859,E2 5991.859} C_VEL
LIN {X 0,Y 482.028,Z 831.81,A -85,B 0,C 180,E1 5995.946,E2 5995.946} C_VEL
LIN {X 0,Y 482.568,Z 832.408,A -85,B 0,C 180,E1 6003.68,E2 6003.68} C_VEL
LIN {X 0,Y 492.32,Z 867.853,A -85,B 0,C 180,E1 6004.645,E2 6004.645} C_VEL
LIN {X 0,Y 491.15,Z 931.622,A -85,B 0,C 180,E1 6006.108,E2 6006.108} C_VEL
LIN {X 0,Y 488.419,Z 983.915,A -85,B 0,C 180,E1 6009.184,E2 6009.184} C_VEL
LIN {X 0,Y 485.901,Z 1026.593,A -85,B 0,C 180,E1 6013.675,E2 6013.675} C_VEL
LIN {X 0,Y 484.26,Z 1057.515,A -85,B 0,C 180,E1 6019.163,E2 6019.163} C_VEL
LIN {X 0,Y 483.37,Z 1075.51,A -85,B 0,C 180,E1 6025.499,E2 6025.499} C_VEL
LIN {X 0,Y 483.25,Z 1078.823,A -85,B 0,C 180,E1 6030.9,E2 6030.9} C_VEL
LIN {X 0,Y 483.271,Z 1070.953,A -85,B 0,C 180,E1 6036.763,E2 6036.763} C_VEL
LIN {X 0,Y 484.059,Z 1050.165,A -85,B 0,C 180,E1 6042.447,E2 6042.447} C_VEL
LIN {X 0,Y 486.15,Z 1016.214,A -85,B 0,C 180,E1 6047.675,E2 6047.675} C_VEL
LIN {X 0,Y 489.248,Z 970.352,A -85,B 0,C 180,E1 6051.85,E2 6051.85} C_VEL
LIN {X 0,Y 491.884,Z 917.768,A -85,B 0,C 180,E1 6054.406,E2 6054.406} C_VEL
LIN {X 0,Y 490.198,Z 855.743,A -85,B 0,C 180,E1 6055.658,E2 6055.658} C_VEL
LIN {X 0,Y 482.674,Z 831.81,A -85,B 0,C 180,E1 6056.484,E2 6056.484} C_VEL
LIN {X 0,Y 482.229,Z 831.81,A -85,B 0,C 180,E1 6066.626,E2 6066.626} C_VEL
LIN {X 0,Y 482.219,Z 831.81,A -85,B 0,C 180,E1 6075.079,E2 6075.079} C_VEL
LIN {X 0,Y 482.075,Z 831.81,A -85,B 0,C 180,E1 6084.378,E2 6084.378} C_VEL
LIN {X 0,Y 482.217,Z 831.81,A -85,B 0,C 180,E1 6093.754,E2 6093.754} C_VEL
LIN {X 0,Y 482.603,Z 831.81,A -85,B 0,C 180,E1 6103.551,E2 6103.551} C_VEL
LIN {X 0,Y 483.151,Z 831.81,A -85,B 0,C 180,E1 6113.686,E2 6113.686} C_VEL
LIN {X 0,Y 483.145,Z 831.81,A -85,B 0,C 180,E1 6122.699,E2 6122.699} C_VEL
LIN {X 0,Y 482.749,Z 831.81,A -85,B 0,C 180,E1 6131.789,E2 6131.789} C_VEL
LIN {X 0,Y 482.576,Z 831.81,A -85,B 0,C 180,E1 6141.924,E2 6141.924} C_VEL
LIN {X 0,Y 482.292,Z 831.81,A -85,B 0,C 180,E1 6151.277,E2 6151.277} C_VEL
LIN {X 0,Y 482.177,Z 831.81,A -85,B 0,C 180,E1 6160.18,E2 6160.18} C_VEL
LIN {X 0,Y 482.084,Z 831.81,A -85,B 0,C 180,E1 6170.466,E2 6170.466} C_VEL
LIN {X 0,Y 482.242,Z 831.81,A -85,B 0,C 180,E1 6180.806,E2 6180.806} C_VEL
LIN {X 0,Y 482.186,Z 831.81,A -85,B 0,C 180,E1 6190.703,E2 6190.703} C_VEL
LIN {X 0,Y 482.818,Z 831.81,A -85,B 0,C 180,E1 6200.045,E2 6200.045} C_VEL
LIN {X 0,Y 483.368,Z 831.81,A -85,B 0,C 180,E1 6209.1,E2 6209.1} C_VEL
LIN {X 0,Y 482.136,Z 832.685,A -85,B 0,C 180,E1 6214.287,E2 6214.287} C_VEL
LIN {X 0,Y 487.401,Z 862.741,A -85,B 0,C 180,E1 6215.919,E2 6215.919} C_VEL
LIN {X 0,Y 485.488,Z 898.094,A -85,B 0,C 180,E1 6219.147,E2 6219.147} C_VEL
LIN {X 0,Y 484.23,Z 922.371,A -85,B 0,C 180,E1 6223.594,E2 6223.594} C_VEL
LIN {X 0,Y 483.821,Z 931.62,A -85,B 0,C 180,E1 6227.336,E2 6227.336} C_VEL
LIN {X 0,Y 483.929,Z 930.948,A -85,B 0,C 180,E1 6233.078,E2 6233.078} C_VEL
LIN {X 0,Y 484.845,Z 915.5,A -85,B 0,C 180,E1 6238.001,E2 6238.001} C_VEL
LIN {X 0,Y 486.411,Z 887.417,A -85,B 0,C 180,E1 6242.045,E2 6242.045} C_VEL
LIN {X 0,Y 486.934,Z 848.879,A -85,B 0,C 180,E1 6244.848,E2 6244.848} C_VEL
LIN {X 0,Y 482.489,Z 831.81,A -85,B 0,C 180,E1 6245.901,E2 6245.901} C_VEL
LIN {X 0,Y 482.119,Z 831.81,A -85,B 0,C 180,E1 6255.09,E2 6255.09} C_VEL
LIN {X 0,Y 482.027,Z 831.81,A -85,B 0,C 180,E1 6264.378,E2 6264.378} C_VEL
LIN {X 0,Y 482.333,Z 831.81,A -85,B 0,C 180,E1 6273.724,E2 6273.724} C_VEL
LIN {X 0,Y 482.57,Z 831.81,A -85,B 0,C 180,E1 6284.497,E2 6284.497} C_VEL
LIN {X 0,Y 482.916,Z 831.81,A -85,B 0,C 180,E1 6293.687,E2 6293.687} C_VEL
LIN {X 0,Y 483,Z 831.81,A -85,B 0,C 180,E1 6300.902,E2 6300.902} C_VEL
LIN {X 0,Y 482.76,Z 831.81,A -85,B 0,C 180,E1 6309.958,E2 6309.958} C_VEL
LIN {X 0,Y 482.622,Z 831.81,A -85,B 0,C 180,E1 6319.281,E2 6319.281} C_VEL
LIN {X 0,Y 482.345,Z 831.81,A -85,B 0,C 180,E1 6329.191,E2 6329.191} C_VEL
LIN {X 0,Y 482.253,Z 831.81,A -85,B 0,C 180,E1 6339.561,E2 6339.561} C_VEL
LIN {X 0,Y 482.165,Z 831.81,A -85,B 0,C 180,E1 6349.819,E2 6349.819} C_VEL
LIN {X 0,Y 482.028,Z 831.81,A -85,B 0,C 180,E1 6355.946,E2 6355.946} C_VEL
LIN {X 0,Y 474.295,Z 831.81,A -85,B 0,C 180,E1 6360.1,E2 6360.1} C_VEL
LIN {X 0,Y 474.661,Z 833.299,A -85,B 0,C 180,E1 6363.321,E2 6363.321} C_VEL
LIN {X 0,Y 484.832,Z 870.189,A -85,B 0,C 180,E1 6364.357,E2 6364.357} C_VEL
LIN {X 0,Y 483.524,Z 931.711,A -85,B 0,C 180,E1 6365.825,E2 6365.825} C_VEL
LIN {X 0,Y 480.617,Z 983.571,A -85,B 0,C 180,E1 6368.952,E2 6368.952} C_VEL
LIN {X 0,Y 477.935,Z 1026.809,A -85,B 0,C 180,E1 6373.633,E2 6373.633} C_VEL
LIN {X 0,Y 476.178,Z 1058.045,A -85,B 0,C 180,E1 6379.441,E2 6379.441} C_VEL
LIN {X 0,Y 475.466,Z 1074.388,A -85,B 0,C 180,E1 6385.424,E2 6385.424} C_VEL
LIN {X 0,Y 475.335,Z 1077.852,A -85,B 0,C 180,E1 6390.915,E2 6390.915} C_VEL
LIN {X 0,Y 475.329,Z 1069.736,A -85,B 0,C 180,E1 6396.876,E2 6396.876} C_VEL
LIN {X 0,Y 476.133,Z 1048.968,A -85,B 0,C 180,E1 6402.637,E2 6402.637} C_VEL
LIN {X 0,Y 478.256,Z 1014.82,A -85,B 0,C 180,E1 6407.965,E2 6407.965} C_VEL
LIN {X 0,Y 481.536,Z 969.672,A -85,B 0,C 180,E1 6412.136,E2 6412.136} C_VEL
LIN {X 0,Y 484.403,Z 916.131,A -85,B 0,C 180,E1 6414.762,E2 6414.762} C_VEL
LIN {X 0,Y 483.078,Z 858.585,A -85,B 0,C 180,E1 6415.932,E2 6415.932} C_VEL
LIN {X 0,Y 474.666,Z 831.81,A -85,B 0,C 180,E1 6416.865,E2 6416.865} C_VEL
LIN {X 0,Y 474.214,Z 831.81,A -85,B 0,C 180,E1 6426.301,E2 6426.301} C_VEL
LIN {X 0,Y 474.093,Z 831.81,A -85,B 0,C 180,E1 6436.506,E2 6436.506} C_VEL
LIN {X 0,Y 474.041,Z 831.81,A -85,B 0,C 180,E1 6445.924,E2 6445.924} C_VEL
LIN {X 0,Y 474.195,Z 831.81,A -85,B 0,C 180,E1 6455.793,E2 6455.793} C_VEL
LIN {X 0,Y 474.654,Z 831.81,A -85,B 0,C 180,E1 6464.228,E2 6464.228} C_VEL
LIN {X 0,Y 475.121,Z 831.81,A -85,B 0,C 180,E1 6473.579,E2 6473.579} C_VEL
LIN {X 0,Y 475.148,Z 831.81,A -85,B 0,C 180,E1 6482.744,E2 6482.744} C_VEL
LIN {X 0,Y 474.727,Z 831.81,A -85,B 0,C 180,E1 6491.991,E2 6491.991} C_VEL
LIN {X 0,Y 474.561,Z 831.81,A -85,B 0,C 180,E1 6501.576,E2 6501.576} C_VEL
LIN {X 0,Y 474.184,Z 831.81,A -85,B 0,C 180,E1 6511.996,E2 6511.996} C_VEL
LIN {X 0,Y 474.083,Z 831.81,A -85,B 0,C 180,E1 6521.215,E2 6521.215} C_VEL
LIN {X 0,Y 474,Z 831.81,A -85,B 0,C 180,E1 6531.368,E2 6531.368} C_VEL
LIN {X 0,Y 474.24,Z 831.81,A -85,B 0,C 180,E1 6541.643,E2 6541.643} C_VEL
LIN {X 0,Y 474.393,Z 831.81,A -85,B 0,C 180,E1 6552.308,E2 6552.308} C_VEL
LIN {X 0,Y 475.014,Z 831.81,A -85,B 0,C 180,E1 6561.734,E2 6561.734} C_VEL
LIN {X 0,Y 474.462,Z 831.81,A -85,B 0,C 180,E1 6570.916,E2 6570.916} C_VEL
LIN {X 0,Y 474.238,Z 833.544,A -85,B 0,C 180,E1 6573.956,E2 6573.956} C_VEL
LIN {X 0,Y 479.813,Z 864.165,A -85,B 0,C 180,E1 6575.672,E2 6575.672} C_VEL
LIN {X 0,Y 477.742,Z 899.606,A -85,B 0,C 180,E1 6578.994,E2 6578.994} C_VEL
LIN {X 0,Y 476.357,Z 924.224,A -85,B 0,C 180,E1 6583.67,E2 6583.67} C_VEL
LIN {X 0,Y 475.899,Z 933.257,A -85,B 0,C 180,E1 6587.634,E2 6587.634} C_VEL
LIN {X 0,Y 475.985,Z 932.852,A -85,B 0,C 180,E1 6592.674,E2 6592.674} C_VEL
LIN {X 0,Y 476.945,Z 918.029,A -85,B 0,C 180,E1 6597.869,E2 6597.869} C_VEL
LIN {X 0,Y 478.632,Z 890.464,A -85,B 0,C 180,E1 6602.082,E2 6602.082} C_VEL
LIN {X 0,Y 479.68,Z 851.915,A -85,B 0,C 180,E1 6605.039,E2 6605.039} C_VEL
LIN {X 0,Y 474.462,Z 831.81,A -85,B 0,C 180,E1 6606.278,E2 6606.278} C_VEL
LIN {X 0,Y 474.065,Z 831.81,A -85,B 0,C 180,E1 6616.508,E2 6616.508} C_VEL
LIN {X 0,Y 474.086,Z 831.81,A -85,B 0,C 180,E1 6625.932,E2 6625.932} C_VEL
LIN {X 0,Y 474.139,Z 831.81,A -85,B 0,C 180,E1 6635.807,E2 6635.807} C_VEL
LIN {X 0,Y 474.457,Z 831.81,A -85,B 0,C 180,E1 6646.121,E2 6646.121} C_VEL
LIN {X 0,Y 474.836,Z 831.81,A -85,B 0,C 180,E1 6655.419,E2 6655.419} C_VEL
LIN {X 0,Y 474.806,Z 831.81,A -85,B 0,C 180,E1 6662.75,E2 6662.75} C_VEL
LIN {X 0,Y 474.839,Z 831.81,A -85,B 0,C 180,E1 6671.992,E2 6671.992} C_VEL
LIN {X 0,Y 474.533,Z 831.81,A -85,B 0,C 180,E1 6681.581,E2 6681.581} C_VEL
LIN {X 0,Y 474.169,Z 831.81,A -85,B 0,C 180,E1 6691.994,E2 6691.994} C_VEL
LIN {X 0,Y 474.153,Z 831.81,A -85,B 0,C 180,E1 6701.226,E2 6701.226} C_VEL
LIN {X 0,Y 474.143,Z 831.81,A -85,B 0,C 180,E1 6711.649,E2 6711.649} C_VEL
LIN {X 0,Y 474.295,Z 831.81,A -85,B 0,C 180,E1 6720.1,E2 6720.1} C_VEL
LIN {X 0,Y 466.476,Z 831.81,A -85,B 0,C 180,E1 6722.864,E2 6722.864} C_VEL
LIN {X 0,Y 477.425,Z 873.192,A -85,B 0,C 180,E1 6724.069,E2 6724.069} C_VEL
LIN {X 0,Y 475.89,Z 932.408,A -85,B 0,C 180,E1 6725.558,E2 6725.558} C_VEL
LIN {X 0,Y 472.826,Z 983.228,A -85,B 0,C 180,E1 6728.711,E2 6728.711} C_VEL
LIN {X 0,Y 470.027,Z 1025.329,A -85,B 0,C 180,E1 6733.349,E2 6733.349} C_VEL
LIN {X 0,Y 468.258,Z 1056.745,A -85,B 0,C 180,E1 6739.261,E2 6739.261} C_VEL
LIN {X 0,Y 467.563,Z 1073.175,A -85,B 0,C 180,E1 6745.346,E2 6745.346} C_VEL
LIN {X 0,Y 467.418,Z 1076.662,A -85,B 0,C 180,E1 6750.93,E2 6750.93} C_VEL
LIN {X 0,Y 467.434,Z 1069.57,A -85,B 0,C 180,E1 6756.525,E2 6756.525} C_VEL
LIN {X 0,Y 468.139,Z 1048.987,A -85,B 0,C 180,E1 6762.582,E2 6762.582} C_VEL
LIN {X 0,Y 470.339,Z 1014.848,A -85,B 0,C 180,E1 6768.093,E2 6768.093} C_VEL
LIN {X 0,Y 473.759,Z 969.986,A -85,B 0,C 180,E1 6772.357,E2 6772.357} C_VEL
LIN {X 0,Y 476.846,Z 916.611,A -85,B 0,C 180,E1 6775.061,E2 6775.061} C_VEL
LIN {X 0,Y 475.488,Z 860.095,A -85,B 0,C 180,E1 6776.255,E2 6776.255} C_VEL
LIN {X 0,Y 466.563,Z 831.81,A -85,B 0,C 180,E1 6777.341,E2 6777.341} C_VEL
LIN {X 0,Y 466.172,Z 831.81,A -85,B 0,C 180,E1 6787.095,E2 6787.095} C_VEL
LIN {X 0,Y 466.025,Z 831.81,A -85,B 0,C 180,E1 6797.112,E2 6797.112} C_VEL
LIN {X 0,Y 466.047,Z 831.81,A -85,B 0,C 180,E1 6807.498,E2 6807.498} C_VEL
LIN {X 0,Y 466.36,Z 831.81,A -85,B 0,C 180,E1 6818.033,E2 6818.033} C_VEL
LIN {X 0,Y 466.833,Z 831.81,A -85,B 0,C 180,E1 6827.799,E2 6827.799} C_VEL
LIN {X 0,Y 466.814,Z 831.81,A -85,B 0,C 180,E1 6837.203,E2 6837.203} C_VEL
LIN {X 0,Y 466.832,Z 831.81,A -85,B 0,C 180,E1 6844.66,E2 6844.66} C_VEL
LIN {X 0,Y 466.734,Z 831.81,A -85,B 0,C 180,E1 6854.113,E2 6854.113} C_VEL
LIN {X 0,Y 466.484,Z 831.81,A -85,B 0,C 180,E1 6863.994,E2 6863.994} C_VEL
LIN {X 0,Y 466.065,Z 831.81,A -85,B 0,C 180,E1 6873.87,E2 6873.87} C_VEL
LIN {X 0,Y 466.011,Z 831.81,A -85,B 0,C 180,E1 6884.439,E2 6884.439} C_VEL
LIN {X 0,Y 466.049,Z 831.81,A -85,B 0,C 180,E1 6895.261,E2 6895.261} C_VEL
LIN {X 0,Y 466.242,Z 831.81,A -85,B 0,C 180,E1 6903.934,E2 6903.934} C_VEL
LIN {X 0,Y 466.49,Z 831.81,A -85,B 0,C 180,E1 6913.947,E2 6913.947} C_VEL
LIN {X 0,Y 466.886,Z 831.81,A -85,B 0,C 180,E1 6923.467,E2 6923.467} C_VEL
LIN {X 0,Y 466.45,Z 831.81,A -85,B 0,C 180,E1 6930.932,E2 6930.932} C_VEL
LIN {X 0,Y 466.154,Z 832.884,A -85,B 0,C 180,E1 6933.558,E2 6933.558} C_VEL
LIN {X 0,Y 472.219,Z 865.605,A -85,B 0,C 180,E1 6935.423,E2 6935.423} C_VEL
LIN {X 0,Y 469.969,Z 901.549,A -85,B 0,C 180,E1 6938.896,E2 6938.896} C_VEL
LIN {X 0,Y 468.551,Z 924.58,A -85,B 0,C 180,E1 6943.318,E2 6943.318} C_VEL
LIN {X 0,Y 467.955,Z 934.821,A -85,B 0,C 180,E1 6947.943,E2 6947.943} C_VEL
LIN {X 0,Y 468.266,Z 932.131,A -85,B 0,C 180,E1 6953.897,E2 6953.897} C_VEL
LIN {X 0,Y 469.518,Z 914.288,A -85,B 0,C 180,E1 6959.053,E2 6959.053} C_VEL
LIN {X 0,Y 471.528,Z 884.5,A -85,B 0,C 180,E1 6963.059,E2 6963.059} C_VEL
LIN {X 0,Y 470.815,Z 847.959,A -85,B 0,C 180,E1 6965.669,E2 6965.669} C_VEL
LIN {X 0,Y 466.403,Z 831.81,A -85,B 0,C 180,E1 6966.558,E2 6966.558} C_VEL
LIN {X 0,Y 465.987,Z 831.81,A -85,B 0,C 180,E1 6977.116,E2 6977.116} C_VEL
LIN {X 0,Y 466.085,Z 831.81,A -85,B 0,C 180,E1 6987.505,E2 6987.505} C_VEL
LIN {X 0,Y 466.131,Z 831.81,A -85,B 0,C 180,E1 6995.987,E2 6995.987} C_VEL
LIN {X 0,Y 466.441,Z 831.81,A -85,B 0,C 180,E1 7005.878,E2 7005.878} C_VEL
LIN {X 0,Y 466.83,Z 831.81,A -85,B 0,C 180,E1 7015.34,E2 7015.34} C_VEL
LIN {X 0,Y 466.807,Z 831.81,A -85,B 0,C 180,E1 7022.797,E2 7022.797} C_VEL
LIN {X 0,Y 466.84,Z 831.81,A -85,B 0,C 180,E1 7032.201,E2 7032.201} C_VEL
LIN {X 0,Y 466.459,Z 831.81,A -85,B 0,C 180,E1 7041.999,E2 7041.999} C_VEL
LIN {X 0,Y 466.124,Z 831.81,A -85,B 0,C 180,E1 7052.497,E2 7052.497} C_VEL
LIN {X 0,Y 466.075,Z 831.81,A -85,B 0,C 180,E1 7062.896,E2 7062.896} C_VEL
LIN {X 0,Y 466.064,Z 831.81,A -85,B 0,C 180,E1 7072.96,E2 7072.96} C_VEL
LIN {X 0,Y 466.476,Z 831.81,A -85,B 0,C 180,E1 7082.864,E2 7082.864} C_VEL
LIN {X 0,Y 471.221,Z 845.207,A -85,B 0,C 180,E1 7083.343,E2 7083.343} C_VEL
LIN {X 0,Y 469.498,Z 866.619,A -85,B 0,C 180,E1 7083.595,E2 7083.595} C_VEL
LIN {X 0,Y 468.487,Z 928.982,A -85,B 0,C 180,E1 7085.108,E2 7085.108} C_VEL
LIN {X 0,Y 465.242,Z 980.759,A -85,B 0,C 180,E1 7088.287,E2 7088.287} C_VEL
LIN {X 0,Y 462.102,Z 1024.172,A -85,B 0,C 180,E1 7093.103,E2 7093.103} C_VEL
LIN {X 0,Y 460.356,Z 1055.445,A -85,B 0,C 180,E1 7099.074,E2 7099.074} C_VEL
LIN {X 0,Y 459.651,Z 1071.96,A -85,B 0,C 180,E1 7105.266,E2 7105.266} C_VEL
LIN {X 0,Y 459.527,Z 1075.474,A -85,B 0,C 180,E1 7110.946,E2 7110.946} C_VEL
LIN {X 0,Y 459.457,Z 1066.976,A -85,B 0,C 180,E1 7117.241,E2 7117.241} C_VEL
LIN {X 0,Y 460.448,Z 1045.058,A -85,B 0,C 180,E1 7123.354,E2 7123.354} C_VEL
LIN {X 0,Y 462.88,Z 1009.388,A -85,B 0,C 180,E1 7128.89,E2 7128.89} C_VEL
LIN {X 0,Y 466.49,Z 962.919,A -85,B 0,C 180,E1 7133.105,E2 7133.105} C_VEL
LIN {X 0,Y 469.532,Z 910.297,A -85,B 0,C 180,E1 7135.571,E2 7135.571} C_VEL
LIN {X 0,Y 467.722,Z 861.106,A -85,B 0,C 180,E1 7136.599,E2 7136.599} C_VEL
LIN {X 0,Y 458.524,Z 831.81,A -85,B 0,C 180,E1 7137.732,E2 7137.732} C_VEL
LIN {X 0,Y 458.083,Z 831.81,A -85,B 0,C 180,E1 7148.869,E2 7148.869} C_VEL
LIN {X 0,Y 457.999,Z 831.81,A -85,B 0,C 180,E1 7158.204,E2 7158.204} C_VEL
LIN {X 0,Y 458.079,Z 831.81,A -85,B 0,C 180,E1 7169.099,E2 7169.099} C_VEL
LIN {X 0,Y 458.444,Z 831.81,A -85,B 0,C 180,E1 7179.658,E2 7179.658} C_VEL
LIN {X 0,Y 458.709,Z 831.81,A -85,B 0,C 180,E1 7189.514,E2 7189.514} C_VEL
LIN {X 0,Y 459.004,Z 831.81,A -85,B 0,C 180,E1 7199.051,E2 7199.051} C_VEL
LIN {X 0,Y 459.057,Z 831.81,A -85,B 0,C 180,E1 7208.554,E2 7208.554} C_VEL
LIN {X 0,Y 458.563,Z 831.81,A -85,B 0,C 180,E1 7218.323,E2 7218.323} C_VEL
LIN {X 0,Y 458.25,Z 831.81,A -85,B 0,C 180,E1 7228.697,E2 7228.697} C_VEL
LIN {X 0,Y 457.952,Z 831.81,A -85,B 0,C 180,E1 7238.855,E2 7238.855} C_VEL
LIN {X 0,Y 457.996,Z 831.81,A -85,B 0,C 180,E1 7248.205,E2 7248.205} C_VEL
LIN {X 0,Y 458.103,Z 831.81,A -85,B 0,C 180,E1 7259.105,E2 7259.105} C_VEL
LIN {X 0,Y 457.999,Z 831.81,A -85,B 0,C 180,E1 7267.601,E2 7267.601} C_VEL
LIN {X 0,Y 458.425,Z 831.81,A -85,B 0,C 180,E1 7277.574,E2 7277.574} C_VEL
LIN {X 0,Y 459.124,Z 831.81,A -85,B 0,C 180,E1 7287.158,E2 7287.158} C_VEL
LIN {X 0,Y 458.321,Z 833.739,A -85,B 0,C 180,E1 7293.206,E2 7293.206} C_VEL
LIN {X 0,Y 464.639,Z 867.482,A -85,B 0,C 180,E1 7295.2,E2 7295.2} C_VEL
LIN {X 0,Y 462.192,Z 903.416,A -85,B 0,C 180,E1 7298.787,E2 7298.787} C_VEL
LIN {X 0,Y 460.625,Z 927.126,A -85,B 0,C 180,E1 7303.613,E2 7303.613} C_VEL
LIN {X 0,Y 460.018,Z 936.335,A -85,B 0,C 180,E1 7308.263,E2 7308.263} C_VEL
LIN {X 0,Y 460.343,Z 934.039,A -85,B 0,C 180,E1 7313.6,E2 7313.6} C_VEL
LIN {X 0,Y 461.597,Z 918.061,A -85,B 0,C 180,E1 7318.716,E2 7318.716} C_VEL
LIN {X 0,Y 463.617,Z 889.883,A -85,B 0,C 180,E1 7322.898,E2 7322.898} C_VEL
LIN {X 0,Y 463.848,Z 851.809,A -85,B 0,C 180,E1 7325.837,E2 7325.837} C_VEL
LIN {X 0,Y 458.339,Z 831.81,A -85,B 0,C 180,E1 7327.03,E2 7327.03} C_VEL
LIN {X 0,Y 457.978,Z 831.81,A -85,B 0,C 180,E1 7337.212,E2 7337.212} C_VEL
LIN {X 0,Y 458.068,Z 831.81,A -85,B 0,C 180,E1 7347.649,E2 7347.649} C_VEL
LIN {X 0,Y 457.984,Z 831.81,A -85,B 0,C 180,E1 7357.602,E2 7357.602} C_VEL
LIN {X 0,Y 458.43,Z 831.81,A -85,B 0,C 180,E1 7367.576,E2 7367.576} C_VEL
LIN {X 0,Y 459.225,Z 831.81,A -85,B 0,C 180,E1 7377.915,E2 7377.915} C_VEL
LIN {X 0,Y 458.862,Z 831.81,A -85,B 0,C 180,E1 7388.561,E2 7388.561} C_VEL
LIN {X 0,Y 458.488,Z 831.81,A -85,B 0,C 180,E1 7398.33,E2 7398.33} C_VEL
LIN {X 0,Y 458.264,Z 831.81,A -85,B 0,C 180,E1 7408.7,E2 7408.7} C_VEL
LIN {X 0,Y 458.075,Z 831.81,A -85,B 0,C 180,E1 7418.875,E2 7418.875} C_VEL
LIN {X 0,Y 457.993,Z 831.81,A -85,B 0,C 180,E1 7428.211,E2 7428.211} C_VEL
LIN {X 0,Y 458.144,Z 831.81,A -85,B 0,C 180,E1 7439.109,E2 7439.109} C_VEL
LIN {X 0,Y 458.493,Z 832.767,A -85,B 0,C 180,E1 7442.505,E2 7442.505} C_VEL
LIN {X 0,Y 469.498,Z 866.619,A -85,B 0,C 180,E1 7443.595,E2 7443.595} C_VEL
LIN {X 0,Y 467.534,Z 883.665,A -85,B 0,C 180,E1 7443.767,E2 7443.767} C_VEL
LIN {X 0,Y 462.28,Z 901.398,A -85,B 0,C 180,E1 7443.875,E2 7443.875} C_VEL
LIN {X 0,Y 459.392,Z 954.698,A -85,B 0,C 180,E1 7446.13,E2 7446.13} C_VEL
LIN {X 0,Y 455.579,Z 1002.183,A -85,B 0,C 180,E1 7450.163,E2 7450.163} C_VEL
LIN {X 0,Y 452.776,Z 1039.818,A -85,B 0,C 180,E1 7455.673,E2 7455.673} C_VEL
LIN {X 0,Y 451.756,Z 1062.164,A -85,B 0,C 180,E1 7461.306,E2 7461.306} C_VEL
LIN {X 0,Y 451.536,Z 1073.051,A -85,B 0,C 180,E1 7467.111,E2 7467.111} C_VEL
LIN {X 0,Y 451.856,Z 1072.126,A -85,B 0,C 180,E1 7473.852,E2 7473.852} C_VEL
LIN {X 0,Y 452.192,Z 1056.118,A -85,B 0,C 180,E1 7480.637,E2 7480.637} C_VEL
LIN {X 0,Y 453.931,Z 1025.572,A -85,B 0,C 180,E1 7486.83,E2 7486.83} C_VEL
LIN {X 0,Y 457.411,Z 982.6,A -85,B 0,C 180,E1 7491.835,E2 7491.835} C_VEL
LIN {X 0,Y 460.917,Z 931.399,A -85,B 0,C 180,E1 7495.137,E2 7495.137} C_VEL
LIN {X 0,Y 462.473,Z 871.451,A -85,B 0,C 180,E1 7496.687,E2 7496.687} C_VEL
LIN {X 0,Y 450.502,Z 831.81,A -85,B 0,C 180,E1 7498.083,E2 7498.083} C_VEL
LIN {X 0,Y 450.072,Z 831.81,A -85,B 0,C 180,E1 7508.593,E2 7508.593} C_VEL
LIN {X 0,Y 449.994,Z 831.81,A -85,B 0,C 180,E1 7519.357,E2 7519.357} C_VEL
LIN {X 0,Y 450.075,Z 831.81,A -85,B 0,C 180,E1 7529.294,E2 7529.294} C_VEL
LIN {X 0,Y 450.371,Z 831.81,A -85,B 0,C 180,E1 7539.277,E2 7539.277} C_VEL
LIN {X 0,Y 450.719,Z 831.81,A -85,B 0,C 180,E1 7549.326,E2 7549.326} C_VEL
LIN {X 0,Y 450.999,Z 831.81,A -85,B 0,C 180,E1 7559.034,E2 7559.034} C_VEL
LIN {X 0,Y 451.026,Z 831.81,A -85,B 0,C 180,E1 7568.707,E2 7568.707} C_VEL
LIN {X 0,Y 450.552,Z 831.81,A -85,B 0,C 180,E1 7578.661,E2 7578.661} C_VEL
LIN {X 0,Y 450.162,Z 831.81,A -85,B 0,C 180,E1 7589.262,E2 7589.262} C_VEL
LIN {X 0,Y 449.935,Z 831.81,A -85,B 0,C 180,E1 7598.607,E2 7598.607} C_VEL
LIN {X 0,Y 449.956,Z 831.81,A -85,B 0,C 180,E1 7608.878,E2 7608.878} C_VEL
LIN {X 0,Y 450.114,Z 831.81,A -85,B 0,C 180,E1 7619.287,E2 7619.287} C_VEL
LIN {X 0,Y 449.961,Z 831.81,A -85,B 0,C 180,E1 7629.26,E2 7629.26} C_VEL
LIN {X 0,Y 450.633,Z 831.81,A -85,B 0,C 180,E1 7639.326,E2 7639.326} C_VEL
LIN {X 0,Y 451.336,Z 831.81,A -85,B 0,C 180,E1 7649.036,E2 7649.036} C_VEL
LIN {X 0,Y 450.181,Z 832.924,A -85,B 0,C 180,E1 7652.777,E2 7652.777} C_VEL
LIN {X 0,Y 457.096,Z 868.093,A -85,B 0,C 180,E1 7654.879,E2 7654.879} C_VEL
LIN {X 0,Y 454.566,Z 903.302,A -85,B 0,C 180,E1 7658.398,E2 7658.398} C_VEL
LIN {X 0,Y 452.825,Z 927.416,A -85,B 0,C 180,E1 7663.216,E2 7663.216} C_VEL
LIN {X 0,Y 452.096,Z 937.78,A -85,B 0,C 180,E1 7668.595,E2 7668.595} C_VEL
LIN {X 0,Y 452.587,Z 934.19,A -85,B 0,C 180,E1 7674.251,E2 7674.251} C_VEL
LIN {X 0,Y 454.021,Z 916.389,A -85,B 0,C 180,E1 7679.494,E2 7679.494} C_VEL
LIN {X 0,Y 456.371,Z 886.675,A -85,B 0,C 180,E1 7683.62,E2 7683.62} C_VEL
LIN {X 0,Y 455.908,Z 851.81,A -85,B 0,C 180,E1 7686.266,E2 7686.266} C_VEL
LIN {X 0,Y 450.224,Z 831.81,A -85,B 0,C 180,E1 7687.617,E2 7687.617} C_VEL
LIN {X 0,Y 449.959,Z 831.81,A -85,B 0,C 180,E1 7696.478,E2 7696.478} C_VEL
LIN {X 0,Y 449.933,Z 831.81,A -85,B 0,C 180,E1 7706.185,E2 7706.185} C_VEL
LIN {X 0,Y 450.098,Z 831.81,A -85,B 0,C 180,E1 7715.075,E2 7715.075} C_VEL
LIN {X 0,Y 450.393,Z 831.81,A -85,B 0,C 180,E1 7725.364,E2 7725.364} C_VEL
LIN {X 0,Y 450.817,Z 831.81,A -85,B 0,C 180,E1 7735.174,E2 7735.174} C_VEL
LIN {X 0,Y 450.826,Z 831.81,A -85,B 0,C 180,E1 7742.896,E2 7742.896} C_VEL
LIN {X 0,Y 450.815,Z 831.81,A -85,B 0,C 180,E1 7752.642,E2 7752.642} C_VEL
LIN {X 0,Y 450.376,Z 831.81,A -85,B 0,C 180,E1 7762.802,E2 7762.802} C_VEL
LIN {X 0,Y 450.123,Z 831.81,A -85,B 0,C 180,E1 7771.509,E2 7771.509} C_VEL
LIN {X 0,Y 450.055,Z 831.81,A -85,B 0,C 180,E1 7781.117,E2 7781.117} C_VEL
LIN {X 0,Y 449.978,Z 831.81,A -85,B 0,C 180,E1 7791.398,E2 7791.398} C_VEL
LIN {X 0,Y 450.446,Z 832.099,A -85,B 0,C 180,E1 7802.054,E2 7802.054} C_VEL
LIN {X 0,Y 462.501,Z 877.055,A -85,B 0,C 180,E1 7803.42,E2 7803.42} C_VEL
LIN {X 0,Y 462.28,Z 901.398,A -85,B 0,C 180,E1 7803.875,E2 7803.875} C_VEL
LIN {X 0,Y 452.974,Z 934.968,A -85,B 0,C 180,E1 7804.729,E2 7804.729} C_VEL
LIN {X 0,Y 449.186,Z 986.135,A -85,B 0,C 180,E1 7808.304,E2 7808.304} C_VEL
LIN {X 0,Y 446.012,Z 1027.386,A -85,B 0,C 180,E1 7813.444,E2 7813.444} C_VEL
LIN {X 0,Y 444.225,Z 1056.339,A -85,B 0,C 180,E1 7819.669,E2 7819.669} C_VEL
LIN {X 0,Y 443.707,Z 1070.831,A -85,B 0,C 180,E1 7826.078,E2 7826.078} C_VEL
LIN {X 0,Y 443.711,Z 1073.096,A -85,B 0,C 180,E1 7830.98,E2 7830.98} C_VEL
LIN {X 0,Y 443.606,Z 1065.924,A -85,B 0,C 180,E1 7836.877,E2 7836.877} C_VEL
LIN {X 0,Y 444.461,Z 1044.924,A -85,B 0,C 180,E1 7843.3,E2 7843.3} C_VEL
LIN {X 0,Y 447.003,Z 1010.384,A -85,B 0,C 180,E1 7849.073,E2 7849.073} C_VEL
LIN {X 0,Y 450.959,Z 964.237,A -85,B 0,C 180,E1 7853.554,E2 7853.554} C_VEL
